C05469=1221.027,359.357,-74.554,-175.932,7.542,148.254
C05470=1221.032,359.109,-74.522,-175.934,7.539,148.254
C05471=1221.036,358.861,-74.489,-175.935,7.537,148.253
C05472=1221.040,358.613,-74.455,-175.937,7.533,148.253
C05473=1221.044,358.365,-74.424,-175.939,7.530,148.253
C05474=1221.048,358.118,-74.390,-175.940,7.528,148.253
C05475=1221.053,357.870,-74.358,-175.941,7.525,148.252
C05476=1221.056,357.622,-74.326,-175.944,7.522,148.252
C05477=1221.061,357.374,-74.293,-175.945,7.519,148.252
C05478=1221.065,357.126,-74.260,-175.947,7.517,148.252
C05479=1221.069,356.878,-74.228,-175.949,7.513,148.251
C05480=1221.073,356.631,-74.195,-175.950,7.510,148.251
C05481=1221.077,356.382,-74.163,-175.952,7.508,148.251
C05482=1221.082,356.135,-74.130,-175.954,7.505,148.251
C05483=1221.086,355.887,-74.098,-175.955,7.502,148.250
C05484=1221.090,355.639,-74.065,-175.957,7.499,148.250
C05485=1221.094,355.391,-74.033,-175.959,7.497,148.250
C05486=1221.098,355.144,-74.000,-175.961,7.493,148.249
C05487=1221.102,354.895,-73.968,-175.962,7.490,148.249
C05488=1221.106,354.648,-73.936,-175.964,7.488,148.249
C05489=1221.110,354.400,-73.903,-175.965,7.485,148.249
C05490=1221.115,354.152,-73.871,-175.967,7.482,148.248
C05491=1221.118,353.905,-73.838,-175.969,7.480,148.248
C05492=1221.123,353.656,-73.806,-175.971,7.477,148.248
C05493=1221.128,353.409,-73.773,-175.972,7.473,148.248
C05494=1221.131,353.161,-73.741,-175.974,7.471,148.247
C05495=1221.136,352.913,-73.708,-175.976,7.468,148.247
C05496=1221.139,352.665,-73.677,-175.978,7.465,148.247
C05497=1221.144,352.417,-73.643,-175.979,7.462,148.247
C05498=1221.148,352.170,-73.612,-175.981,7.460,148.247
C05499=1221.152,351.921,-73.580,-175.983,7.457,148.246
C05500=1221.156,351.674,-73.546,-175.985,7.454,148.246
C05501=1221.160,351.426,-73.515,-175.987,7.452,148.246
C05502=1221.165,351.178,-73.482,-175.988,7.448,148.246
C05503=1221.169,350.930,-73.451,-175.990,7.445,148.245
C05504=1221.173,350.682,-73.417,-175.992,7.443,148.245
C05505=1221.177,350.434,-73.386,-175.994,7.439,148.245
C05506=1221.182,350.186,-73.354,-175.995,7.437,148.245
C05507=1221.185,349.938,-73.322,-175.997,7.434,148.245
C05508=1221.190,349.691,-73.289,-175.999,7.431,148.244
C05509=1221.193,349.443,-73.257,-176.001,7.429,148.244
C05510=1221.198,349.195,-73.225,-176.002,7.426,148.244
C05511=1221.202,348.947,-73.193,-176.005,7.423,148.244
C05512=1221.206,348.699,-73.160,-176.006,7.420,148.244
C05513=1221.210,348.451,-73.128,-176.008,7.418,148.244
C05514=1221.215,348.204,-73.096,-176.010,7.414,148.243
C05515=1221.219,347.955,-73.064,-176.012,7.412,148.243
C05516=1221.223,347.707,-73.031,-176.013,7.409,148.243
C05517=1221.227,347.460,-73.000,-176.016,7.406,148.243
C05518=1221.232,347.211,-72.967,-176.017,7.403,148.243
C05519=1221.236,346.963,-72.936,-176.019,7.401,148.242
C05520=1221.240,346.716,-72.904,-176.021,7.397,148.242
C05521=1221.244,346.468,-72.872,-176.023,7.395,148.242
C05522=1221.248,346.220,-72.840,-176.024,7.392,148.242
C05523=1221.253,345.972,-72.808,-176.027,7.389,148.242
C05524=1221.257,345.724,-72.776,-176.029,7.387,148.242
C05525=1221.260,345.476,-72.744,-176.031,7.383,148.241
C05526=1221.265,345.229,-72.711,-176.032,7.381,148.241
C05527=1221.269,344.981,-72.679,-176.034,7.378,148.241
C05528=1221.274,344.732,-72.648,-176.036,7.375,148.241
C05529=1221.278,344.485,-72.616,-176.038,7.372,148.241
C05530=1221.282,344.237,-72.584,-176.040,7.370,148.240
C05531=1221.286,343.988,-72.552,-176.042,7.367,148.240
C05532=1221.290,343.741,-72.520,-176.043,7.364,148.240
C05533=1221.294,343.493,-72.489,-176.045,7.362,148.240
C05534=1221.299,343.244,-72.456,-176.048,7.358,148.240
C05535=1221.303,342.997,-72.425,-176.049,7.356,148.240
C05536=1221.307,342.749,-72.393,-176.051,7.353,148.239
C05537=1221.312,342.501,-72.361,-176.053,7.350,148.239
C05538=1221.315,342.253,-72.329,-176.055,7.348,148.239
C05539=1221.319,342.005,-72.297,-176.057,7.345,148.239
C05540=1221.324,341.758,-72.265,-176.059,7.342,148.239
C05541=1221.329,341.480,-72.230,-176.061,7.339,148.239
C05542=1221.333,341.202,-72.195,-176.063,7.335,148.238
C05543=1221.338,340.924,-72.158,-176.066,7.333,148.238
C05544=1221.343,340.646,-72.123,-176.068,7.330,148.238
C05545=1221.346,340.398,-72.092,-176.070,7.326,148.238
C05546=1221.351,340.151,-72.060,-176.072,7.324,148.238
C05547=1221.355,339.902,-72.028,-176.074,7.322,148.238
C05548=1221.360,339.654,-71.997,-176.076,7.318,148.238
C05549=1221.363,339.406,-71.965,-176.077,7.316,148.237
C05550=1221.367,339.158,-71.933,-176.079,7.313,148.237
C05551=1221.371,338.911,-71.902,-176.082,7.310,148.237
C05552=1221.376,338.662,-71.870,-176.083,7.308,148.237
C05553=1221.381,338.415,-71.839,-176.086,7.304,148.237
C05554=1221.384,338.167,-71.807,-176.088,7.302,148.237
C05555=1221.389,337.919,-71.776,-176.089,7.299,148.237
C05556=1221.393,337.671,-71.744,-176.091,7.296,148.236
C05557=1221.398,337.423,-71.712,-176.093,7.294,148.236
C05558=1221.402,337.174,-71.681,-176.096,7.291,148.236
C05559=1221.406,336.927,-71.649,-176.097,7.288,148.236
C05560=1221.410,336.679,-71.618,-176.099,7.286,148.236
C05561=1221.414,336.431,-71.587,-176.102,7.282,148.236
C05562=1221.418,336.183,-71.555,-176.103,7.280,148.236
C05563=1221.422,335.935,-71.523,-176.106,7.277,148.236
C05564=1221.426,335.687,-71.492,-176.108,7.274,148.236
C05565=1221.431,335.439,-71.460,-176.109,7.272,148.235
C05566=1221.435,335.191,-71.429,-176.112,7.269,148.235
C05567=1221.439,334.943,-71.397,-176.114,7.266,148.235
C05568=1221.444,334.695,-71.367,-176.116,7.263,148.235
C05569=1221.447,334.447,-71.335,-176.118,7.261,148.235
C05570=1221.452,334.199,-71.304,-176.119,7.258,148.235
C05571=1221.456,333.951,-71.272,-176.122,7.255,148.235
C05572=1221.460,333.703,-71.241,-176.124,7.253,148.235
C05573=1221.465,333.455,-71.210,-176.126,7.249,148.234
C05574=1221.469,333.207,-71.179,-176.128,7.247,148.234
C05575=1221.473,332.959,-71.147,-176.130,7.244,148.234
C05576=1221.477,332.711,-71.116,-176.132,7.241,148.234
C05577=1221.481,332.463,-71.085,-176.134,7.239,148.234
C05578=1221.485,332.215,-71.053,-176.137,7.236,148.234
C05579=1221.490,331.967,-71.022,-176.138,7.233,148.234
C05580=1221.494,331.719,-70.991,-176.140,7.231,148.234
C05581=1221.498,331.471,-70.960,-176.143,7.228,148.234
C05582=1221.503,331.223,-70.929,-176.145,7.225,148.234
C05583=1221.507,330.975,-70.898,-176.147,7.222,148.234
C05584=1221.511,330.727,-70.866,-176.149,7.220,148.234
C05585=1221.515,330.479,-70.835,-176.151,7.217,148.233
C05586=1221.519,330.231,-70.804,-176.153,7.214,148.233
C05587=1221.523,329.983,-70.772,-176.155,7.212,148.233
C05588=1221.528,329.735,-70.742,-176.158,7.209,148.233
C05589=1221.532,329.487,-70.711,-176.159,7.206,148.233
C05590=1221.536,329.239,-70.679,-176.161,7.204,148.233
C05591=1221.541,328.991,-70.648,-176.163,7.201,148.233
C05592=1221.545,328.742,-70.617,-176.166,7.198,148.233
C05593=1221.549,328.494,-70.587,-176.168,7.195,148.233
C05594=1221.553,328.247,-70.555,-176.170,7.193,148.233
C05595=1221.557,327.998,-70.524,-176.172,7.190,148.232
C05596=1221.562,327.750,-70.493,-176.174,7.187,148.233
C05597=1221.566,327.503,-70.463,-176.176,7.185,148.232
C05598=1221.570,327.255,-70.431,-176.178,7.182,148.232
C05599=1221.574,327.007,-70.400,-176.181,7.179,148.232
C05600=1221.579,326.759,-70.369,-176.183,7.176,148.232
C05601=1221.582,326.510,-70.339,-176.185,7.174,148.232
C05602=1221.587,326.262,-70.308,-176.187,7.171,148.232
C05603=1221.592,326.014,-70.277,-176.189,7.168,148.232
C05604=1221.595,325.766,-70.245,-176.191,7.166,148.232
C05605=1221.600,325.518,-70.215,-176.193,7.163,148.232
C05606=1221.603,325.270,-70.184,-176.196,7.161,148.232
C05607=1221.608,325.022,-70.153,-176.197,7.158,148.232
C05608=1221.612,324.774,-70.123,-176.200,7.155,148.232
C05609=1221.617,324.526,-70.092,-176.202,7.153,148.232
C05610=1221.621,324.277,-70.061,-176.204,7.149,148.232
C05611=1221.625,324.030,-70.031,-176.206,7.147,148.232
C05612=1221.630,323.782,-70.000,-176.208,7.145,148.232
C05613=1221.634,323.533,-69.969,-176.211,7.142,148.231
C05614=1221.638,323.285,-69.938,-176.213,7.139,148.231
C05615=1221.642,323.038,-69.908,-176.215,7.136,148.231
C05616=1221.646,322.789,-69.877,-176.217,7.134,148.231
C05617=1221.651,322.541,-69.846,-176.220,7.131,148.231
C05618=1221.655,322.293,-69.816,-176.222,7.129,148.231
C05619=1221.659,322.045,-69.785,-176.223,7.126,148.231
C05620=1221.663,321.797,-69.754,-176.226,7.123,148.231
C05621=1221.668,321.549,-69.723,-176.228,7.121,148.231
C05622=1221.672,321.301,-69.693,-176.231,7.118,148.231
C05623=1221.676,321.053,-69.662,-176.232,7.115,148.231
C05624=1221.680,320.804,-69.631,-176.235,7.113,148.231
C05625=1221.684,320.557,-69.601,-176.237,7.110,148.231
C05626=1221.689,320.309,-69.570,-176.239,7.107,148.231
C05627=1221.693,320.061,-69.539,-176.241,7.104,148.231
C05628=1221.697,319.813,-69.509,-176.244,7.102,148.231
C05629=1221.702,319.564,-69.479,-176.246,7.100,148.231
C05630=1221.705,319.316,-69.448,-176.248,7.097,148.231
C05631=1221.710,319.068,-69.418,-176.250,7.094,148.231
C05632=1221.714,318.820,-69.387,-176.253,7.091,148.231
C05633=1221.718,318.572,-69.356,-176.255,7.089,148.231
C05634=1221.723,318.323,-69.326,-176.257,7.087,148.231
C05635=1221.727,318.076,-69.296,-176.259,7.083,148.231
C05636=1221.731,317.828,-69.265,-176.261,7.081,148.231
C05637=1221.735,317.579,-69.234,-176.264,7.078,148.231
C05638=1221.739,317.332,-69.204,-176.266,7.076,148.231
C05639=1221.744,317.083,-69.174,-176.268,7.073,148.231
C05640=1221.748,316.835,-69.144,-176.270,7.070,148.231
C05641=1221.753,316.587,-69.113,-176.272,7.068,148.231
C05642=1221.756,316.338,-69.083,-176.275,7.065,148.231
C05643=1221.761,316.090,-69.053,-176.277,7.063,148.231
C05644=1221.765,315.843,-69.022,-176.280,7.060,148.231
C05645=1221.770,315.566,-68.989,-176.281,7.057,148.231
C05646=1221.775,315.291,-68.955,-176.284,7.054,148.231
C05647=1221.780,315.015,-68.922,-176.287,7.051,148.231
C05648=1221.784,314.739,-68.888,-176.289,7.048,148.231
C05649=1221.788,314.492,-68.858,-176.291,7.046,148.231
C05650=1221.793,314.243,-68.827,-176.294,7.044,148.231
C05651=1221.796,313.995,-68.797,-176.296,7.041,148.231
C05652=1221.801,313.746,-68.767,-176.298,7.038,148.231
C05653=1221.805,313.499,-68.737,-176.301,7.035,148.231
C05654=1221.810,313.250,-68.707,-176.303,7.033,148.231
C05655=1221.814,313.002,-68.677,-176.305,7.031,148.231
C05656=1221.819,312.754,-68.646,-176.307,7.028,148.231
C05657=1221.823,312.506,-68.616,-176.310,7.025,148.231
C05658=1221.827,312.259,-68.586,-176.312,7.022,148.231
C05659=1221.832,312.010,-68.556,-176.314,7.020,148.231
C05660=1221.835,311.762,-68.526,-176.316,7.018,148.231
C05661=1221.840,311.513,-68.495,-176.319,7.015,148.231
C05662=1221.844,311.265,-68.466,-176.321,7.013,148.231
C05663=1221.848,311.017,-68.436,-176.324,7.010,148.231
C05664=1221.853,310.769,-68.406,-176.326,7.007,148.231
C05665=1221.857,310.521,-68.376,-176.328,7.005,148.231
C05666=1221.861,310.272,-68.346,-176.330,7.002,148.231
C05667=1221.865,310.025,-68.315,-176.332,7.000,148.231
C05668=1221.870,309.776,-68.286,-176.335,6.997,148.231
C05669=1221.874,309.528,-68.256,-176.337,6.994,148.231
C05670=1221.878,309.280,-68.226,-176.339,6.992,148.231
C05671=1221.883,309.032,-68.196,-176.342,6.989,148.231
C05672=1221.887,308.784,-68.166,-176.344,6.987,148.231
C05673=1221.891,308.536,-68.136,-176.346,6.985,148.231
C05674=1221.896,308.287,-68.107,-176.349,6.982,148.231
C05675=1221.900,308.039,-68.077,-176.351,6.979,148.231
C05676=1221.904,307.791,-68.046,-176.354,6.976,148.231
C05677=1221.908,307.543,-68.017,-176.356,6.974,148.231
C05678=1221.913,307.295,-67.988,-176.358,6.972,148.231
C05679=1221.917,307.047,-67.957,-176.360,6.969,148.231
C05680=1221.921,306.798,-67.927,-176.363,6.967,148.231
C05681=1221.926,306.550,-67.898,-176.365,6.964,148.231
C05682=1221.930,306.302,-67.868,-176.367,6.961,148.231
C05683=1221.934,306.054,-67.838,-176.369,6.959,148.231
C05684=1221.939,305.806,-67.808,-176.372,6.956,148.231
C05685=1221.943,305.557,-67.779,-176.374,6.954,148.231
C05686=1221.947,305.309,-67.749,-176.376,6.952,148.231
C05687=1221.951,305.061,-67.720,-176.379,6.949,148.231
C05688=1221.956,304.813,-67.689,-176.381,6.946,148.231
C05689=1221.960,304.565,-67.660,-176.384,6.943,148.231
C05690=1221.964,304.316,-67.630,-176.386,6.941,148.232
C05691=1221.968,304.068,-67.601,-176.388,6.939,148.232
C05692=1221.972,303.820,-67.571,-176.391,6.936,148.232
C05693=1221.977,303.571,-67.541,-176.393,6.934,148.232
C05694=1221.982,303.323,-67.512,-176.395,6.932,148.232
C05695=1221.986,303.075,-67.482,-176.398,6.929,148.232
C05696=1221.990,302.826,-67.453,-176.400,6.927,148.232
C05697=1221.995,302.579,-67.424,-176.403,6.923,148.232
C05698=1221.999,302.331,-67.394,-176.405,6.921,148.232
C05699=1222.003,302.083,-67.364,-176.407,6.919,148.232
C05700=1222.007,301.835,-67.335,-176.410,6.916,148.232
C05701=1222.012,301.586,-67.305,-176.412,6.914,148.232
C05702=1222.016,301.338,-67.275,-176.414,6.912,148.232
C05703=1222.020,301.090,-67.246,-176.417,6.909,148.232
C05704=1222.024,300.841,-67.216,-176.419,6.906,148.232
C05705=1222.029,300.593,-67.187,-176.421,6.904,148.233
C05706=1222.033,300.344,-67.158,-176.424,6.901,148.233
C05707=1222.038,300.097,-67.129,-176.426,6.899,148.233
C05708=1222.042,299.848,-67.100,-176.428,6.897,148.233
C05709=1222.046,299.600,-67.070,-176.431,6.894,148.233
C05710=1222.050,299.352,-67.041,-176.433,6.892,148.233
C05711=1222.055,299.104,-67.011,-176.436,6.889,148.233
C05712=1222.059,298.855,-66.982,-176.438,6.886,148.233
C05713=1222.063,298.607,-66.952,-176.440,6.885,148.233
C05714=1222.068,298.359,-66.923,-176.443,6.881,148.233
C05715=1222.072,298.111,-66.894,-176.445,6.879,148.233
C05716=1222.076,297.862,-66.865,-176.447,6.877,148.233
C05717=1222.081,297.614,-66.836,-176.450,6.874,148.233
C05718=1222.085,297.366,-66.806,-176.452,6.872,148.233
C05719=1222.089,297.117,-66.777,-176.454,6.870,148.233
C05720=1222.094,296.870,-66.748,-176.457,6.867,148.234
C05721=1222.098,296.621,-66.719,-176.459,6.865,148.234
C05722=1222.102,296.373,-66.689,-176.462,6.862,148.234
C05723=1222.107,296.124,-66.660,-176.464,6.859,148.234
C05724=1222.111,295.876,-66.630,-176.466,6.857,148.234
C05725=1222.115,295.628,-66.603,-176.469,6.855,148.234
C05726=1222.119,295.380,-66.573,-176.472,6.852,148.234
C05727=1222.124,295.132,-66.544,-176.474,6.850,148.234
C05728=1222.128,294.884,-66.514,-176.476,6.848,148.234
C05729=1222.132,294.635,-66.486,-176.478,6.845,148.234
C05730=1222.137,294.387,-66.456,-176.481,6.843,148.235
C05731=1222.141,294.139,-66.427,-176.483,6.841,148.235
C05732=1222.146,293.890,-66.398,-176.486,6.838,148.235
C05733=1222.149,293.642,-66.369,-176.488,6.835,148.235
C05734=1222.154,293.394,-66.340,-176.490,6.833,148.235
C05735=1222.158,293.146,-66.312,-176.493,6.830,148.235
C05736=1222.163,292.897,-66.282,-176.495,6.828,148.235
C05737=1222.167,292.648,-66.253,-176.497,6.826,148.235
C05738=1222.172,292.401,-66.224,-176.500,6.823,148.235
C05739=1222.175,292.153,-66.195,-176.503,6.821,148.235
C05740=1222.180,291.904,-66.167,-176.505,6.819,148.235
C05741=1222.184,291.656,-66.137,-176.507,6.816,148.235
C05742=1222.189,291.408,-66.109,-176.510,6.814,148.236
C05743=1222.193,291.159,-66.079,-176.512,6.812,148.236
C05744=1222.197,290.911,-66.051,-176.515,6.809,148.236
C05745=1222.202,290.663,-66.022,-176.517,6.806,148.236
C05746=1222.206,290.414,-65.993,-176.519,6.804,148.236
C05747=1222.210,290.166,-65.964,-176.522,6.802,148.236
C05748=1222.215,289.918,-65.936,-176.524,6.799,148.236
C05749=1222.220,289.644,-65.905,-176.527,6.796,148.236
C05750=1222.224,289.370,-65.872,-176.530,6.794,148.237
C05751=1222.229,289.096,-65.841,-176.532,6.791,148.237
C05752=1222.234,288.821,-65.809,-176.535,6.789,148.237
C05753=1222.238,288.573,-65.780,-176.538,6.786,148.237
C05754=1222.243,288.325,-65.751,-176.540,6.784,148.237
C05755=1222.247,288.076,-65.723,-176.542,6.782,148.237
C05756=1222.251,287.828,-65.694,-176.545,6.779,148.237
C05757=1222.256,287.580,-65.665,-176.547,6.777,148.237
C05758=1222.260,287.331,-65.637,-176.549,6.775,148.237
C05759=1222.264,287.083,-65.608,-176.552,6.772,148.238
C05760=1222.269,286.835,-65.579,-176.554,6.770,148.238
C05761=1222.273,286.586,-65.551,-176.557,6.768,148.238
C05762=1222.277,286.339,-65.522,-176.559,6.766,148.238
C05763=1222.282,286.090,-65.493,-176.562,6.763,148.238
C05764=1222.286,285.841,-65.465,-176.564,6.761,148.238
C05765=1222.291,285.594,-65.436,-176.567,6.759,148.238
C05766=1222.294,285.345,-65.408,-176.569,6.756,148.238
C05767=1222.299,285.096,-65.379,-176.571,6.753,148.238
C05768=1222.304,284.848,-65.351,-176.574,6.751,148.239
C05769=1222.308,284.599,-65.323,-176.576,6.749,148.239
C05770=1222.312,284.352,-65.294,-176.579,6.746,148.239
C05771=1222.316,284.103,-65.265,-176.581,6.744,148.239
C05772=1222.321,283.855,-65.237,-176.583,6.742,148.239
C05773=1222.325,283.606,-65.209,-176.586,6.739,148.239
C05774=1222.329,283.358,-65.180,-176.589,6.737,148.240
C05775=1222.334,283.110,-65.151,-176.591,6.735,148.240
C05776=1222.338,282.861,-65.123,-176.593,6.733,148.240
C05777=1222.343,282.613,-65.095,-176.596,6.730,148.240
C05778=1222.347,282.365,-65.066,-176.598,6.728,148.240
C05779=1222.352,282.116,-65.038,-176.601,6.726,148.240
C05780=1222.356,281.868,-65.010,-176.603,6.724,148.240
C05781=1222.361,281.620,-64.981,-176.606,6.721,148.240
C05782=1222.364,281.371,-64.953,-176.608,6.719,148.241
C05783=1222.370,281.123,-64.925,-176.610,6.717,148.241
C05784=1222.373,280.874,-64.897,-176.613,6.714,148.241
C05785=1222.377,280.626,-64.869,-176.616,6.712,148.241
C05786=1222.382,280.378,-64.840,-176.618,6.709,148.241
C05787=1222.386,280.129,-64.812,-176.620,6.708,148.241
C05788=1222.391,279.881,-64.784,-176.623,6.705,148.241
C05789=1222.395,279.632,-64.756,-176.626,6.703,148.242
C05790=1222.400,279.384,-64.727,-176.628,6.700,148.242
C05791=1222.404,279.135,-64.699,-176.630,6.698,148.242
C05792=1222.408,278.888,-64.671,-176.633,6.695,148.242
C05793=1222.412,278.639,-64.643,-176.635,6.693,148.242
C05794=1222.417,278.391,-64.615,-176.638,6.691,148.242
C05795=1222.421,278.142,-64.586,-176.640,6.689,148.243
C05796=1222.426,277.894,-64.558,-176.643,6.686,148.243
C05797=1222.430,277.646,-64.531,-176.645,6.684,148.243
C05798=1222.434,277.397,-64.502,-176.647,6.682,148.243
C05799=1222.439,277.149,-64.474,-176.650,6.680,148.243
C05800=1222.443,276.901,-64.446,-176.652,6.677,148.243
C05801=1222.448,276.652,-64.418,-176.655,6.675,148.244
C05802=1222.452,276.403,-64.390,-176.657,6.673,148.244
C05803=1222.456,276.156,-64.362,-176.660,6.671,148.244
C05804=1222.461,275.907,-64.334,-176.662,6.669,148.244
C05805=1222.465,275.659,-64.306,-176.665,6.666,148.244
C05806=1222.469,275.411,-64.278,-176.667,6.664,148.244
C05807=1222.474,275.161,-64.250,-176.670,6.662,148.245
C05808=1222.478,274.914,-64.222,-176.672,6.660,148.245
C05809=1222.482,274.665,-64.194,-176.675,6.657,148.245
C05810=1222.486,274.417,-64.166,-176.677,6.655,148.245
C05811=1222.491,274.168,-64.138,-176.679,6.653,148.245
C05812=1222.496,273.920,-64.111,-176.682,6.651,148.245
C05813=1222.500,273.672,-64.083,-176.685,6.648,148.245
C05814=1222.504,273.423,-64.055,-176.687,6.646,148.246
C05815=1222.509,273.175,-64.027,-176.689,6.644,148.246
C05816=1222.513,272.927,-63.999,-176.692,6.642,148.246
C05817=1222.517,272.678,-63.971,-176.694,6.640,148.246
C05818=1222.522,272.430,-63.944,-176.697,6.637,148.246
C05819=1222.526,272.181,-63.916,-176.699,6.635,148.246
C05820=1222.531,271.933,-63.887,-176.702,6.633,148.247
C05821=1222.535,271.684,-63.860,-176.704,6.631,148.247
C05822=1222.539,271.436,-63.832,-176.707,6.629,148.247
C05823=1222.544,271.187,-63.805,-176.709,6.626,148.247
C05824=1222.548,270.939,-63.777,-176.712,6.624,148.247
C05825=1222.553,270.690,-63.749,-176.714,6.622,148.247
C05826=1222.557,270.442,-63.722,-176.717,6.620,148.248
C05827=1222.562,270.194,-63.694,-176.719,6.618,148.248
C05828=1222.566,269.945,-63.666,-176.722,6.615,148.248
C05829=1222.570,269.697,-63.639,-176.724,6.613,148.248
C05830=1222.575,269.449,-63.612,-176.727,6.611,148.248
C05831=1222.578,269.200,-63.583,-176.729,6.609,148.249
C05832=1222.583,268.951,-63.556,-176.731,6.607,148.249
C05833=1222.588,268.703,-63.528,-176.735,6.604,148.249
C05834=1222.592,268.454,-63.501,-176.737,6.602,148.249
C05835=1222.597,268.206,-63.473,-176.739,6.600,148.249
C05836=1222.601,267.958,-63.446,-176.741,6.598,148.250
C05837=1222.606,267.710,-63.418,-176.744,6.596,148.250
C05838=1222.610,267.461,-63.391,-176.747,6.593,148.250
C05839=1222.614,267.212,-63.363,-176.749,6.591,148.250
C05840=1222.619,266.964,-63.336,-176.751,6.589,148.250
C05841=1222.623,266.716,-63.309,-176.754,6.587,148.251
C05842=1222.627,266.467,-63.280,-176.756,6.585,148.251
C05843=1222.632,266.219,-63.253,-176.759,6.583,148.251
C05844=1222.636,265.970,-63.226,-176.762,6.580,148.251
C05845=1222.641,265.722,-63.199,-176.764,6.578,148.251
C05846=1222.645,265.473,-63.171,-176.767,6.576,148.252
C05847=1222.649,265.225,-63.144,-176.769,6.574,148.252
C05848=1222.654,264.977,-63.116,-176.771,6.572,148.252
C05849=1222.658,264.728,-63.089,-176.773,6.570,148.252
C05850=1222.663,264.479,-63.062,-176.777,6.567,148.252
C05851=1222.667,264.231,-63.034,-176.779,6.565,148.253
C05852=1222.672,263.983,-63.007,-176.781,6.563,148.253
C05853=1222.677,263.710,-62.977,-176.784,6.561,148.253
C05854=1222.682,263.437,-62.948,-176.787,6.558,148.253
C05855=1222.686,263.165,-62.918,-176.789,6.556,148.253
C05856=1222.691,262.891,-62.887,-176.792,6.553,148.254
C05857=1222.695,262.643,-62.860,-176.795,6.551,148.254
C05858=1222.700,262.395,-62.832,-176.797,6.549,148.254
C05859=1222.704,262.147,-62.805,-176.800,6.547,148.254
C05860=1222.709,261.898,-62.778,-176.802,6.545,148.255
C05861=1222.712,261.649,-62.751,-176.804,6.543,148.255
C05862=1222.717,261.401,-62.724,-176.808,6.540,148.255
C05863=1222.722,261.152,-62.697,-176.810,6.538,148.255
C05864=1222.726,260.904,-62.670,-176.812,6.536,148.255
C05865=1222.731,260.656,-62.643,-176.815,6.534,148.256
C05866=1222.735,260.407,-62.615,-176.817,6.532,148.256
C05867=1222.740,260.159,-62.588,-176.820,6.530,148.256
C05868=1222.743,259.910,-62.562,-176.822,6.528,148.256
C05869=1222.748,259.662,-62.535,-176.825,6.526,148.256
C05870=1222.753,259.413,-62.507,-176.828,6.524,148.257
C05871=1222.757,259.165,-62.480,-176.830,6.521,148.257
C05872=1222.762,258.916,-62.453,-176.832,6.520,148.257
C05873=1222.766,258.668,-62.427,-176.835,6.518,148.257
C05874=1222.771,258.419,-62.400,-176.837,6.515,148.257
C05875=1222.775,258.171,-62.373,-176.840,6.514,148.258
C05876=1222.779,257.922,-62.345,-176.842,6.512,148.258
C05877=1222.784,257.673,-62.318,-176.845,6.509,148.258
C05878=1222.788,257.425,-62.292,-176.848,6.507,148.258
C05879=1222.793,257.176,-62.265,-176.850,6.505,148.258
C05880=1222.797,256.928,-62.238,-176.852,6.503,148.259
C05881=1222.802,256.679,-62.211,-176.855,6.501,148.259
C05882=1222.806,256.431,-62.184,-176.857,6.499,148.259
C05883=1222.810,256.183,-62.157,-176.860,6.497,148.259
C05884=1222.815,255.934,-62.130,-176.862,6.495,148.260
C05885=1222.820,255.686,-62.103,-176.865,6.492,148.260
C05886=1222.824,255.438,-62.076,-176.868,6.490,148.260
C05887=1222.829,255.189,-62.050,-176.870,6.488,148.260
C05888=1222.833,254.939,-62.023,-176.872,6.486,148.260
C05889=1222.837,254.691,-61.996,-176.875,6.484,148.261
C05890=1222.841,254.443,-61.969,-176.878,6.482,148.261
C05891=1222.846,254.194,-61.942,-176.880,6.480,148.261
C05892=1222.850,253.946,-61.916,-176.882,6.478,148.261
C05893=1222.855,253.697,-61.889,-176.885,6.476,148.262
C05894=1222.859,253.448,-61.862,-176.887,6.474,148.262
C05895=1222.863,253.200,-61.836,-176.890,6.472,148.262
C05896=1222.868,252.952,-61.809,-176.893,6.469,148.262
C05897=1222.872,252.703,-61.783,-176.895,6.467,148.262
C05898=1222.877,252.454,-61.756,-176.898,6.465,148.263
C05899=1222.882,252.206,-61.729,-176.900,6.463,148.263
C05900=1222.885,251.958,-61.702,-176.903,6.462,148.263
C05901=1222.890,251.709,-61.676,-176.905,6.459,148.263
C05902=1222.894,251.460,-61.650,-176.908,6.457,148.264
C05903=1222.899,251.212,-61.622,-176.910,6.456,148.264
C05904=1222.904,250.963,-61.596,-176.912,6.453,148.264
C05905=1222.908,250.715,-61.570,-176.915,6.452,148.264
C05906=1222.913,250.466,-61.543,-176.917,6.450,148.265
C05907=1222.917,250.217,-61.517,-176.920,6.447,148.265
C05908=1222.921,249.969,-61.490,-176.923,6.445,148.265
C05909=1222.925,249.721,-61.463,-176.925,6.443,148.265
C05910=1222.930,249.471,-61.437,-176.928,6.441,148.266
C05911=1222.935,249.224,-61.411,-176.930,6.439,148.266
C05912=1222.939,248.976,-61.384,-176.933,6.437,148.266
C05913=1222.944,248.727,-61.358,-176.935,6.435,148.266
C05914=1222.948,248.478,-61.331,-176.938,6.433,148.267
C05915=1222.953,248.229,-61.305,-176.940,6.431,148.267
C05916=1222.957,247.981,-61.278,-176.943,6.429,148.267
C05917=1222.961,247.732,-61.252,-176.945,6.427,148.267
C05918=1222.966,247.484,-61.225,-176.947,6.425,148.268
C05919=1222.970,247.235,-61.200,-176.950,6.423,148.268
C05920=1222.975,246.986,-61.173,-176.953,6.421,148.268
C05921=1222.979,246.738,-61.147,-176.955,6.419,148.269
C05922=1222.984,246.489,-61.120,-176.957,6.417,148.269
C05923=1222.988,246.240,-61.094,-176.960,6.415,148.269
C05924=1222.993,245.993,-61.068,-176.963,6.413,148.269
C05925=1222.998,245.744,-61.042,-176.966,6.411,148.269
C05926=1223.002,245.495,-61.015,-176.968,6.409,148.270
C05927=1223.006,245.246,-60.989,-176.971,6.407,148.270
C05928=1223.010,244.998,-60.962,-176.973,6.405,148.270
C05929=1223.015,244.749,-60.937,-176.976,6.403,148.271
C05930=1223.020,244.500,-60.910,-176.978,6.401,148.271
C05931=1223.024,244.252,-60.884,-176.981,6.399,148.271
C05932=1223.028,244.004,-60.858,-176.983,6.397,148.271
C05933=1223.033,243.755,-60.832,-176.986,6.395,148.272
C05934=1223.037,243.507,-60.806,-176.988,6.393,148.272
C05935=1223.042,243.258,-60.779,-176.991,6.391,148.272
C05936=1223.046,243.009,-60.753,-176.993,6.389,148.272
C05937=1223.050,242.761,-60.727,-176.996,6.387,148.273
C05938=1223.055,242.512,-60.702,-176.998,6.385,148.273
C05939=1223.060,242.263,-60.675,-177.001,6.383,148.273
C05940=1223.064,242.015,-60.649,-177.003,6.381,148.273
C05941=1223.068,241.766,-60.623,-177.006,6.380,148.274
C05942=1223.073,241.517,-60.597,-177.008,6.378,148.274
C05943=1223.077,241.268,-60.571,-177.011,6.375,148.274
C05944=1223.082,241.021,-60.545,-177.013,6.374,148.274
C05945=1223.087,240.772,-60.518,-177.016,6.372,148.275
C05946=1223.091,240.523,-60.493,-177.018,6.370,148.275
C05947=1223.095,240.274,-60.467,-177.021,6.368,148.275
C05948=1223.100,240.026,-60.442,-177.023,6.366,148.275
C05949=1223.105,239.778,-60.415,-177.026,6.364,148.276
C05950=1223.109,239.529,-60.389,-177.028,6.362,148.276
C05951=1223.113,239.280,-60.363,-177.031,6.360,148.276
C05952=1223.118,239.031,-60.337,-177.034,6.358,148.277
C05953=1223.122,238.783,-60.312,-177.036,6.356,148.277
C05954=1223.127,238.534,-60.286,-177.038,6.354,148.277
C05955=1223.131,238.286,-60.259,-177.041,6.352,148.277
C05956=1223.135,238.037,-60.233,-177.044,6.351,148.278
C05957=1223.141,237.766,-60.206,-177.047,6.348,148.278
C05958=1223.145,237.494,-60.178,-177.049,6.346,148.278
C05959=1223.150,237.223,-60.149,-177.052,6.344,148.279
C05960=1223.155,236.951,-60.121,-177.055,6.342,148.279
C05961=1223.159,236.703,-60.095,-177.057,6.340,148.279
C05962=1223.165,236.454,-60.069,-177.059,6.338,148.279
C05963=1223.169,236.205,-60.044,-177.062,6.336,148.280
C05964=1223.173,235.957,-60.018,-177.065,6.334,148.280
C05965=1223.178,235.708,-59.993,-177.067,6.333,148.280
C05966=1223.182,235.460,-59.967,-177.070,6.331,148.281
C05967=1223.187,235.211,-59.941,-177.073,6.329,148.281
C05968=1223.191,234.962,-59.915,-177.075,6.327,148.281
C05969=1223.196,234.714,-59.890,-177.077,6.325,148.281
C05970=1223.200,234.465,-59.864,-177.080,6.323,148.282
C05971=1223.205,234.216,-59.838,-177.083,6.321,148.282
C05972=1223.210,233.968,-59.812,-177.085,6.319,148.282
C05973=1223.214,233.719,-59.787,-177.088,6.317,148.283
C05974=1223.218,233.470,-59.761,-177.090,6.315,148.283
C05975=1223.223,233.222,-59.736,-177.093,6.313,148.283
C05976=1223.228,232.973,-59.711,-177.095,6.311,148.283
C05977=1223.232,232.724,-59.685,-177.098,6.309,148.284
C05978=1223.237,232.476,-59.659,-177.100,6.308,148.284
C05979=1223.241,232.227,-59.634,-177.103,6.306,148.284
C05980=1223.245,231.978,-59.608,-177.106,6.304,148.285
C05981=1223.250,231.730,-59.583,-177.108,6.302,148.285
C05982=1223.254,231.481,-59.557,-177.110,6.300,148.285
C05983=1223.259,231.233,-59.532,-177.113,6.298,148.285
C05984=1223.263,230.984,-59.506,-177.116,6.296,148.286
C05985=1223.268,230.735,-59.481,-177.118,6.294,148.286
C05986=1223.272,230.487,-59.455,-177.121,6.292,148.286
C05987=1223.277,230.237,-59.430,-177.124,6.290,148.287
C05988=1223.282,229.989,-59.405,-177.126,6.289,148.287
C05989=1223.286,229.741,-59.379,-177.128,6.286,148.287
C05990=1223.290,229.492,-59.353,-177.131,6.285,148.287
C05991=1223.295,229.243,-59.329,-177.134,6.283,148.288
C05992=1223.299,228.995,-59.303,-177.136,6.281,148.288
C05993=1223.304,228.746,-59.278,-177.139,6.279,148.288
C05994=1223.308,228.497,-59.253,-177.141,6.278,148.289
C05995=1223.312,228.248,-59.227,-177.143,6.276,148.289
C05996=1223.317,228.000,-59.202,-177.146,6.274,148.289
C05997=1223.322,227.751,-59.177,-177.149,6.272,148.290
C05998=1223.327,227.503,-59.151,-177.151,6.270,148.290
C05999=1223.331,227.254,-59.126,-177.154,6.268,148.290
C06000=1223.336,227.005,-59.101,-177.156,6.266,148.290
C06001=1223.340,226.757,-59.076,-177.159,6.265,148.291
C06002=1223.344,226.508,-59.051,-177.161,6.263,148.291
C06003=1223.349,226.259,-59.025,-177.164,6.261,148.291
C06004=1223.353,226.010,-59.000,-177.167,6.259,148.292
C06005=1223.358,225.762,-58.975,-177.169,6.257,148.292
C06006=1223.362,225.513,-58.949,-177.172,6.255,148.292
C06007=1223.367,225.264,-58.925,-177.175,6.253,148.293
C06008=1223.371,225.015,-58.899,-177.177,6.252,148.293
C06009=1223.376,224.767,-58.875,-177.179,6.249,148.293
C06010=1223.380,224.518,-58.849,-177.182,6.247,148.293
C06011=1223.386,224.269,-58.824,-177.185,6.246,148.294
C06012=1223.389,224.021,-58.799,-177.187,6.245,148.294
C06013=1223.394,223.772,-58.775,-177.189,6.243,148.294
C06014=1223.398,223.523,-58.749,-177.192,6.241,148.295
C06015=1223.404,223.274,-58.724,-177.194,6.239,148.295
C06016=1223.407,223.026,-58.699,-177.197,6.237,148.295
C06017=1223.412,222.777,-58.674,-177.200,6.235,148.296
C06018=1223.416,222.528,-58.649,-177.202,6.233,148.296
C06019=1223.422,222.280,-58.624,-177.205,6.232,148.296
C06020=1223.426,222.031,-58.600,-177.208,6.230,148.297
C06021=1223.430,221.783,-58.574,-177.210,6.228,148.297
C06022=1223.435,221.534,-58.549,-177.213,6.226,148.297
C06023=1223.439,221.285,-58.524,-177.216,6.224,148.298
C06024=1223.444,221.037,-58.500,-177.218,6.222,148.298
C06025=1223.448,220.787,-58.475,-177.220,6.221,148.298
C06026=1223.452,220.539,-58.450,-177.222,6.219,148.299
C06027=1223.457,220.290,-58.425,-177.225,6.217,148.299
C06028=1223.462,220.041,-58.400,-177.228,6.215,148.299
C06029=1223.466,219.793,-58.375,-177.230,6.213,148.300
C06030=1223.471,219.544,-58.350,-177.233,6.212,148.300
C06031=1223.476,219.295,-58.326,-177.236,6.210,148.300
C06032=1223.480,219.046,-58.301,-177.238,6.208,148.300
C06033=1223.485,218.798,-58.276,-177.241,6.206,148.301
C06034=1223.489,218.549,-58.251,-177.243,6.204,148.301
C06035=1223.493,218.300,-58.227,-177.246,6.202,148.301
C06036=1223.499,218.052,-58.202,-177.249,6.200,148.302
C06037=1223.502,217.803,-58.177,-177.251,6.199,148.302
C06038=1223.507,217.554,-58.152,-177.253,6.198,148.303
C06039=1223.512,217.306,-58.127,-177.256,6.196,148.303
C06040=1223.516,217.056,-58.103,-177.259,6.194,148.303
C06041=1223.521,216.808,-58.078,-177.261,6.192,148.303
C06042=1223.525,216.559,-58.053,-177.264,6.190,148.304
C06043=1223.530,216.311,-58.029,-177.267,6.188,148.304
C06044=1223.534,216.062,-58.004,-177.269,6.186,148.304
C06045=1223.539,215.813,-57.979,-177.272,6.185,148.305
C06046=1223.543,215.564,-57.955,-177.274,6.183,148.305
C06047=1223.548,215.316,-57.931,-177.276,6.182,148.306
C06048=1223.553,215.066,-57.906,-177.279,6.180,148.306
C06049=1223.557,214.818,-57.882,-177.282,6.178,148.306
C06050=1223.562,214.570,-57.856,-177.284,6.176,148.307
C06051=1223.566,214.320,-57.832,-177.287,6.174,148.307
C06052=1223.571,214.072,-57.807,-177.290,6.172,148.307
C06053=1223.575,213.823,-57.783,-177.292,6.171,148.308
C06054=1223.579,213.574,-57.759,-177.295,6.169,148.308
C06055=1223.584,213.326,-57.734,-177.298,6.167,148.308
C06056=1223.589,213.077,-57.710,-177.300,6.166,148.309
C06057=1223.594,212.828,-57.685,-177.302,6.164,148.309
C06058=1223.598,212.579,-57.661,-177.305,6.162,148.309
C06059=1223.603,212.331,-57.636,-177.308,6.160,148.310
C06060=1223.607,212.082,-57.612,-177.310,6.158,148.310
C06061=1223.612,211.811,-57.586,-177.313,6.157,148.310
C06062=1223.617,211.540,-57.559,-177.315,6.155,148.311
C06063=1223.622,211.270,-57.532,-177.319,6.153,148.311
C06064=1223.627,211.000,-57.506,-177.321,6.151,148.311
C06065=1223.632,210.752,-57.481,-177.324,6.149,148.312
C06066=1223.636,210.503,-57.457,-177.326,6.148,148.312
C06067=1223.641,210.253,-57.433,-177.329,6.146,148.312
C06068=1223.645,210.005,-57.409,-177.332,6.144,148.313
C06069=1223.650,209.756,-57.385,-177.334,6.142,148.313
C06070=1223.654,209.507,-57.360,-177.337,6.140,148.313
C06071=1223.659,209.259,-57.336,-177.340,6.138,148.314
C06072=1223.663,209.010,-57.312,-177.342,6.137,148.314
C06073=1223.668,208.761,-57.287,-177.344,6.136,148.314
C06074=1223.672,208.512,-57.263,-177.347,6.134,148.315
C06075=1223.677,208.263,-57.239,-177.350,6.132,148.315
C06076=1223.682,208.015,-57.215,-177.352,6.130,148.315
C06077=1223.686,207.766,-57.190,-177.355,6.128,148.316
C06078=1223.691,207.518,-57.166,-177.357,6.127,148.316
C06079=1223.696,207.268,-57.142,-177.360,6.125,148.317
C06080=1223.700,207.019,-57.118,-177.362,6.123,148.317
C06081=1223.704,206.771,-57.094,-177.365,6.122,148.317
C06082=1223.709,206.522,-57.070,-177.367,6.120,148.318
C06083=1223.714,206.273,-57.046,-177.370,6.118,148.318
C06084=1223.718,206.024,-57.021,-177.373,6.116,148.318
C06085=1223.722,205.776,-56.997,-177.375,6.115,148.319
C06086=1223.728,205.526,-56.973,-177.378,6.113,148.319
C06087=1223.732,205.278,-56.949,-177.381,6.112,148.319
C06088=1223.737,205.029,-56.925,-177.383,6.110,148.320
C06089=1223.741,204.780,-56.902,-177.386,6.108,148.320
C06090=1223.745,204.531,-56.877,-177.388,6.107,148.321
C06091=1223.750,204.283,-56.853,-177.391,6.105,148.321
C06092=1223.755,204.034,-56.829,-177.393,6.103,148.321
C06093=1223.759,203.785,-56.805,-177.396,6.101,148.322
C06094=1223.764,203.536,-56.782,-177.399,6.099,148.322
C06095=1223.768,203.288,-56.758,-177.401,6.098,148.322
C06096=1223.774,203.039,-56.733,-177.403,6.097,148.323
C06097=1223.778,202.790,-56.710,-177.406,6.095,148.323
C06098=1223.782,202.541,-56.685,-177.409,6.093,148.323
C06099=1223.787,202.292,-56.662,-177.412,6.091,148.324
C06100=1223.791,202.043,-56.638,-177.414,6.090,148.324
C06101=1223.796,201.794,-56.615,-177.416,6.089,148.325
C06102=1223.800,201.546,-56.591,-177.419,6.087,148.325
C06103=1223.806,201.297,-56.567,-177.422,6.085,148.325
C06104=1223.810,201.048,-56.543,-177.424,6.083,148.326
C06105=1223.815,200.799,-56.519,-177.427,6.081,148.326
C06106=1223.819,200.551,-56.495,-177.429,6.080,148.326
C06107=1223.824,200.302,-56.472,-177.432,6.078,148.327
C06108=1223.828,200.053,-56.447,-177.434,6.076,148.327
C06109=1223.832,199.804,-56.424,-177.437,6.075,148.327
C06110=1223.837,199.555,-56.400,-177.440,6.073,148.328
C06111=1223.841,199.306,-56.377,-177.442,6.072,148.328
C06112=1223.846,199.058,-56.352,-177.445,6.070,148.329
C06113=1223.851,198.809,-56.329,-177.447,6.068,148.329
C06114=1223.855,198.560,-56.306,-177.450,6.066,148.329
C06115=1223.860,198.311,-56.282,-177.453,6.065,148.330
C06116=1223.864,198.062,-56.258,-177.455,6.064,148.330
C06117=1223.869,197.813,-56.235,-177.457,6.062,148.330
C06118=1223.873,197.565,-56.211,-177.460,6.060,148.331
C06119=1223.879,197.315,-56.187,-177.463,6.058,148.331
C06120=1223.883,197.067,-56.163,-177.465,6.057,148.332
C06121=1223.888,196.818,-56.139,-177.468,6.056,148.332
C06122=1223.892,196.569,-56.117,-177.471,6.054,148.332
C06123=1223.897,196.320,-56.093,-177.473,6.052,148.333
C06124=1223.901,196.072,-56.069,-177.476,6.050,148.333
C06125=1223.906,195.823,-56.046,-177.478,6.049,148.333
C06126=1223.910,195.574,-56.023,-177.481,6.047,148.334
C06127=1223.915,195.325,-55.998,-177.483,6.045,148.334
C06128=1223.920,195.076,-55.975,-177.486,6.043,148.334
C06129=1223.924,194.827,-55.952,-177.488,6.043,148.335
C06130=1223.929,194.578,-55.928,-177.491,6.041,148.335
C06131=1223.934,194.329,-55.905,-177.494,6.039,148.336
C06132=1223.938,194.081,-55.881,-177.496,6.037,148.336
C06133=1223.943,193.832,-55.858,-177.498,6.036,148.336
C06134=1223.947,193.583,-55.834,-177.501,6.034,148.337
C06135=1223.952,193.334,-55.811,-177.504,6.033,148.337
C06136=1223.957,193.085,-55.788,-177.507,6.031,148.338
C06137=1223.961,192.836,-55.763,-177.509,6.030,148.338
C06138=1223.965,192.588,-55.741,-177.512,6.028,148.338
C06139=1223.970,192.338,-55.717,-177.514,6.026,148.339
C06140=1223.975,192.090,-55.694,-177.517,6.025,148.339
C06141=1223.980,191.841,-55.671,-177.519,6.024,148.339
C06142=1223.985,191.592,-55.648,-177.522,6.022,148.340
C06143=1223.989,191.343,-55.624,-177.524,6.020,148.340
C06144=1223.994,191.094,-55.601,-177.527,6.018,148.341
C06145=1223.998,190.845,-55.578,-177.529,6.017,148.341
C06146=1224.003,190.596,-55.555,-177.532,6.015,148.341
C06147=1224.007,190.347,-55.531,-177.535,6.014,148.342
C06148=1224.012,190.099,-55.507,-177.537,6.012,148.342
C06149=1224.016,189.850,-55.484,-177.539,6.011,148.343
C06150=1224.021,189.602,-55.462,-177.543,6.009,148.343
C06151=1224.026,189.353,-55.438,-177.545,6.007,148.343
C06152=1224.030,189.104,-55.415,-177.547,6.006,148.344
C06153=1224.035,188.855,-55.392,-177.550,6.005,148.344
C06154=1224.040,188.606,-55.368,-177.553,6.003,148.345
C06155=1224.044,188.356,-55.346,-177.555,6.001,148.345
C06156=1224.049,188.107,-55.323,-177.558,6.000,148.345
C06157=1224.053,187.858,-55.299,-177.560,5.998,148.346
C06158=1224.059,187.610,-55.276,-177.563,5.997,148.346
C06159=1224.063,187.361,-55.254,-177.565,5.996,148.347
C06160=1224.067,187.112,-55.230,-177.568,5.994,148.347
C06161=1224.072,186.863,-55.207,-177.571,5.992,148.347
C06162=1224.076,186.614,-55.184,-177.574,5.990,148.348
C06163=1224.081,186.365,-55.161,-177.576,5.989,148.348
C06164=1224.086,186.117,-55.138,-177.578,5.988,148.349
C06165=1224.090,185.847,-55.113,-177.581,5.986,148.349
C06166=1224.095,185.577,-55.088,-177.584,5.984,148.349
C06167=1224.101,185.307,-55.063,-177.587,5.982,148.350
C06168=1224.105,185.038,-55.039,-177.589,5.980,148.350
C06169=1224.111,184.790,-55.016,-177.592,5.980,148.351
C06170=1224.115,184.541,-54.992,-177.595,5.978,148.351
C06171=1224.120,184.291,-54.970,-177.597,5.976,148.352
C06172=1224.124,184.042,-54.947,-177.599,5.975,148.352
C06173=1224.129,183.793,-54.923,-177.602,5.973,148.352
C06174=1224.134,183.545,-54.901,-177.605,5.972,148.353
C06175=1224.138,183.296,-54.878,-177.608,5.970,148.353
C06176=1224.142,183.047,-54.856,-177.610,5.969,148.354
C06177=1224.147,182.798,-54.832,-177.613,5.967,148.354
C06178=1224.152,182.549,-54.809,-177.615,5.965,148.354
C06179=1224.156,182.301,-54.786,-177.617,5.964,148.355
C06180=1224.161,182.051,-54.764,-177.620,5.963,148.355
C06181=1224.165,181.802,-54.741,-177.623,5.961,148.356
C06182=1224.170,181.553,-54.718,-177.625,5.960,148.356
C06183=1224.176,181.304,-54.695,-177.628,5.958,148.356
C06184=1224.180,181.056,-54.673,-177.631,5.957,148.357
C06185=1224.184,180.807,-54.649,-177.633,5.956,148.357
C06186=1224.189,180.557,-54.627,-177.636,5.954,148.358
C06187=1224.194,180.309,-54.604,-177.638,5.952,148.358
C06188=1224.198,180.060,-54.582,-177.640,5.951,148.358
C06189=1224.203,179.810,-54.559,-177.644,5.949,148.359
C06190=1224.207,179.562,-54.536,-177.646,5.948,148.359
C06191=1224.212,179.313,-54.514,-177.648,5.947,148.360
C06192=1224.216,179.064,-54.491,-177.651,5.945,148.360
C06193=1224.221,178.814,-54.468,-177.654,5.943,148.360
C06194=1224.226,178.566,-54.446,-177.656,5.942,148.361
C06195=1224.231,178.317,-54.423,-177.659,5.940,148.361
C06196=1224.235,178.068,-54.401,-177.662,5.939,148.362
C06197=1224.240,177.820,-54.378,-177.664,5.938,148.362
C06198=1224.245,177.570,-54.356,-177.667,5.936,148.363
C06199=1224.249,177.321,-54.332,-177.669,5.934,148.363
C06200=1224.254,177.073,-54.311,-177.672,5.933,148.363
C06201=1224.258,176.824,-54.288,-177.674,5.931,148.364
C06202=1224.263,176.574,-54.265,-177.677,5.931,148.364
C06203=1224.268,176.326,-54.243,-177.679,5.929,148.365
C06204=1224.273,176.077,-54.220,-177.682,5.927,148.365
C06205=1224.277,175.828,-54.197,-177.684,5.926,148.365
C06206=1224.282,175.579,-54.175,-177.687,5.925,148.366
C06207=1224.286,175.330,-54.153,-177.690,5.923,148.366
C06208=1224.290,175.081,-54.130,-177.692,5.922,148.367
C06209=1224.296,174.832,-54.108,-177.695,5.920,148.367
C06210=1224.300,174.583,-54.085,-177.698,5.918,148.368
C06211=1224.305,174.335,-54.063,-177.700,5.917,148.368
C06212=1224.310,174.085,-54.041,-177.703,5.916,148.368
C06213=1224.314,173.836,-54.018,-177.705,5.915,148.369
C06214=1224.319,173.587,-53.996,-177.708,5.913,148.369
C06215=1224.324,173.338,-53.974,-177.710,5.911,148.370
C06216=1224.328,173.090,-53.951,-177.713,5.910,148.370
C06217=1224.333,172.840,-53.929,-177.715,5.908,148.371
C06218=1224.338,172.591,-53.907,-177.718,5.908,148.371
C06219=1224.342,172.343,-53.884,-177.720,5.906,148.372
C06220=1224.346,172.094,-53.862,-177.723,5.904,148.372
C06221=1224.352,171.845,-53.840,-177.725,5.903,148.372
C06222=1224.356,171.596,-53.817,-177.728,5.902,148.373
C06223=1224.360,171.347,-53.795,-177.731,5.900,148.373
C06224=1224.366,171.098,-53.773,-177.733,5.899,148.374
C06225=1224.370,170.848,-53.751,-177.736,5.897,148.374
C06226=1224.375,170.600,-53.728,-177.738,5.896,148.375
C06227=1224.379,170.351,-53.706,-177.741,5.894,148.375
C06228=1224.385,170.102,-53.684,-177.744,5.893,148.375
C06229=1224.389,169.853,-53.662,-177.746,5.892,148.376
C06230=1224.393,169.605,-53.640,-177.749,5.890,148.376
C06231=1224.398,169.355,-53.618,-177.751,5.889,148.377
C06232=1224.403,169.106,-53.595,-177.754,5.887,148.377
C06233=1224.408,168.857,-53.573,-177.757,5.886,148.378
C06234=1224.412,168.608,-53.551,-177.759,5.885,148.378
C06235=1224.417,168.359,-53.530,-177.762,5.883,148.378
C06236=1224.422,168.109,-53.507,-177.764,5.882,148.379
C06237=1224.426,167.861,-53.484,-177.767,5.881,148.379
C06238=1224.431,167.612,-53.462,-177.769,5.879,148.380
C06239=1224.435,167.363,-53.441,-177.772,5.878,148.380
C06240=1224.440,167.114,-53.419,-177.775,5.876,148.381
C06241=1224.445,166.865,-53.397,-177.777,5.875,148.381
C06242=1224.450,166.616,-53.374,-177.779,5.873,148.381
C06243=1224.454,166.367,-53.353,-177.782,5.873,148.382
C06244=1224.459,166.118,-53.331,-177.785,5.871,148.382
C06245=1224.464,165.869,-53.309,-177.787,5.869,148.383
C06246=1224.468,165.620,-53.287,-177.789,5.868,148.383
C06247=1224.473,165.371,-53.265,-177.793,5.867,148.384
C06248=1224.478,165.122,-53.244,-177.795,5.866,148.384
C06249=1224.482,164.873,-53.222,-177.797,5.864,148.385
C06250=1224.487,164.624,-53.199,-177.800,5.863,148.385
C06251=1224.492,164.375,-53.177,-177.803,5.861,148.385
C06252=1224.497,164.126,-53.156,-177.805,5.859,148.386
C06253=1224.501,163.877,-53.133,-177.808,5.859,148.386
C06254=1224.506,163.628,-53.112,-177.810,5.857,148.387
C06255=1224.510,163.379,-53.090,-177.813,5.856,148.387
C06256=1224.515,163.130,-53.068,-177.816,5.854,148.388
C06257=1224.520,162.882,-53.046,-177.818,5.853,148.388
C06258=1224.524,162.632,-53.024,-177.821,5.852,148.389
C06259=1224.529,162.384,-53.003,-177.823,5.851,148.389
C06260=1224.533,162.134,-52.981,-177.826,5.849,148.390
C06261=1224.538,161.886,-52.959,-177.828,5.847,148.390
C06262=1224.542,161.636,-52.937,-177.831,5.847,148.391
C06263=1224.547,161.387,-52.916,-177.834,5.845,148.391
C06264=1224.552,161.138,-52.894,-177.836,5.844,148.391
C06265=1224.557,160.889,-52.872,-177.839,5.842,148.392
C06266=1224.561,160.640,-52.850,-177.841,5.841,148.392
C06267=1224.566,160.391,-52.828,-177.844,5.840,148.393
C06268=1224.571,160.142,-52.807,-177.846,5.839,148.393
C06269=1224.576,159.873,-52.783,-177.849,5.837,148.394
C06270=1224.582,159.604,-52.760,-177.852,5.836,148.394
C06271=1224.586,159.335,-52.737,-177.855,5.834,148.395
C06272=1224.591,159.066,-52.713,-177.857,5.833,148.395
C06273=1224.596,158.817,-52.692,-177.860,5.831,148.396
C06274=1224.601,158.568,-52.669,-177.862,5.830,148.396
C06275=1224.606,158.319,-52.648,-177.865,5.829,148.397
C06276=1224.610,158.069,-52.626,-177.867,5.828,148.397
C06277=1224.614,157.821,-52.605,-177.870,5.826,148.397
C06278=1224.619,157.572,-52.584,-177.873,5.825,148.398
C06279=1224.624,157.322,-52.562,-177.875,5.824,148.398
C06280=1224.628,157.074,-52.541,-177.877,5.823,148.399
C06281=1224.633,156.825,-52.519,-177.881,5.821,148.399
C06282=1224.638,156.575,-52.498,-177.883,5.819,148.400
C06283=1224.643,156.326,-52.476,-177.886,5.819,148.400
C06284=1224.648,156.078,-52.454,-177.888,5.817,148.401
C06285=1224.653,155.829,-52.433,-177.891,5.816,148.401
C06286=1224.656,155.580,-52.412,-177.894,5.814,148.402
C06287=1224.661,155.331,-52.390,-177.896,5.813,148.402
C06288=1224.666,155.082,-52.369,-177.898,5.812,148.402
C06289=1224.671,154.832,-52.347,-177.901,5.811,148.403
C06290=1224.676,154.583,-52.326,-177.904,5.809,148.403
C06291=1224.681,154.334,-52.305,-177.906,5.808,148.404
C06292=1224.685,154.086,-52.283,-177.909,5.807,148.404
C06293=1224.689,153.836,-52.262,-177.911,5.806,148.405
C06294=1224.694,153.587,-52.240,-177.914,5.804,148.405
C06295=1224.699,153.338,-52.219,-177.916,5.803,148.406
C06296=1224.704,153.089,-52.197,-177.919,5.801,148.406
C06297=1224.709,152.840,-52.176,-177.922,5.801,148.407
C06298=1224.713,152.591,-52.155,-177.924,5.799,148.407
C06299=1224.718,152.342,-52.134,-177.926,5.798,148.408
C06300=1224.722,152.093,-52.112,-177.929,5.796,148.408
C06301=1224.728,151.843,-52.091,-177.932,5.795,148.409
C06302=1224.732,151.595,-52.070,-177.935,5.794,148.409
C06303=1224.737,151.346,-52.049,-177.937,5.793,148.410
C06304=1224.742,151.097,-52.028,-177.939,5.792,148.410
C06305=1224.746,150.847,-52.006,-177.942,5.790,148.411
C06306=1224.751,150.599,-51.985,-177.944,5.789,148.411
C06307=1224.756,150.350,-51.964,-177.947,5.788,148.412
C06308=1224.761,150.100,-51.943,-177.949,5.787,148.412
C06309=1224.764,149.851,-51.922,-177.952,5.785,148.412
C06310=1224.770,149.602,-51.901,-177.955,5.785,148.413
C06311=1224.774,149.353,-51.879,-177.957,5.783,148.413
C06312=1224.780,149.104,-51.858,-177.960,5.782,148.414
C06313=1224.784,148.855,-51.838,-177.963,5.780,148.414
C06314=1224.788,148.606,-51.816,-177.965,5.779,148.415
C06315=1224.794,148.357,-51.795,-177.968,5.778,148.415
C06316=1224.798,148.108,-51.774,-177.970,5.777,148.416
C06317=1224.803,147.859,-51.753,-177.973,5.775,148.416
C06318=1224.808,147.610,-51.732,-177.975,5.774,148.417
C06319=1224.812,147.361,-51.711,-177.978,5.773,148.417
C06320=1224.817,147.112,-51.689,-177.981,5.772,148.418
C06321=1224.821,146.863,-51.669,-177.983,5.771,148.418
C06322=1224.826,146.613,-51.648,-177.986,5.769,148.419
C06323=1224.831,146.365,-51.626,-177.988,5.768,148.419
C06324=1224.836,146.116,-51.606,-177.991,5.767,148.420
C06325=1224.841,145.866,-51.585,-177.993,5.766,148.420
C06326=1224.846,145.617,-51.564,-177.996,5.764,148.420
C06327=1224.849,145.368,-51.543,-177.998,5.764,148.421
C06328=1224.855,145.119,-51.522,-178.001,5.762,148.421
C06329=1224.859,144.870,-51.501,-178.004,5.761,148.422
C06330=1224.864,144.621,-51.480,-178.006,5.760,148.423
C06331=1224.868,144.372,-51.459,-178.009,5.758,148.423
C06332=1224.874,144.123,-51.438,-178.011,5.758,148.424
C06333=1224.878,143.874,-51.418,-178.014,5.756,148.424
C06334=1224.883,143.625,-51.397,-178.016,5.755,148.425
C06335=1224.888,143.375,-51.376,-178.019,5.753,148.425
C06336=1224.892,143.126,-51.355,-178.022,5.753,148.426
C06337=1224.897,142.877,-51.334,-178.024,5.751,148.426
C06338=1224.902,142.628,-51.313,-178.027,5.750,148.427
C06339=1224.907,142.379,-51.292,-178.029,5.749,148.427
C06340=1224.911,142.130,-51.272,-178.032,5.748,148.427
C06341=1224.916,141.881,-51.251,-178.034,5.747,148.428
C06342=1224.921,141.632,-51.230,-178.037,5.745,148.428
C06343=1224.926,141.383,-51.209,-178.040,5.744,148.429
C06344=1224.930,141.134,-51.189,-178.042,5.743,148.429
C06345=1224.936,140.885,-51.168,-178.045,5.742,148.430
C06346=1224.940,140.636,-51.148,-178.047,5.741,148.430
C06347=1224.944,140.387,-51.127,-178.050,5.740,148.431
C06348=1224.949,140.137,-51.105,-178.052,5.739,148.431
C06349=1224.953,139.888,-51.085,-178.055,5.737,148.432
C06350=1224.958,139.639,-51.064,-178.057,5.736,148.432
C06351=1224.963,139.390,-51.044,-178.060,5.735,148.433
C06352=1224.968,139.141,-51.023,-178.063,5.734,148.433
C06353=1224.972,138.892,-51.002,-178.065,5.733,148.434
C06354=1224.977,138.643,-50.982,-178.068,5.731,148.434
C06355=1224.982,138.394,-50.961,-178.070,5.730,148.435
C06356=1224.987,138.144,-50.941,-178.073,5.730,148.435
C06357=1224.992,137.895,-50.920,-178.075,5.728,148.436
C06358=1224.996,137.646,-50.900,-178.078,5.727,148.436
C06359=1225.001,137.397,-50.880,-178.081,5.725,148.437
C06360=1225.006,137.148,-50.859,-178.083,5.725,148.437
C06361=1225.010,136.899,-50.838,-178.085,5.724,148.438
C06362=1225.016,136.650,-50.817,-178.088,5.722,148.438
C06363=1225.020,136.401,-50.797,-178.091,5.721,148.439
C06364=1225.024,136.152,-50.777,-178.093,5.719,148.439
C06365=1225.030,135.902,-50.756,-178.096,5.719,148.440
C06366=1225.034,135.653,-50.735,-178.098,5.718,148.440
C06367=1225.039,135.404,-50.716,-178.101,5.716,148.441
C06368=1225.044,135.155,-50.695,-178.103,5.715,148.441
C06369=1225.048,134.906,-50.674,-178.106,5.714,148.442
C06370=1225.053,134.657,-50.654,-178.109,5.713,148.442
C06371=1225.059,134.408,-50.633,-178.111,5.712,148.443
C06372=1225.063,134.159,-50.613,-178.114,5.711,148.443
C06373=1225.067,133.890,-50.591,-178.116,5.710,148.444
C06374=1225.073,133.621,-50.569,-178.120,5.708,148.445
C06375=1225.078,133.353,-50.547,-178.122,5.707,148.445
C06376=1225.084,133.084,-50.525,-178.125,5.706,148.446
C06377=1225.088,132.835,-50.505,-178.128,5.705,148.446
C06378=1225.093,132.586,-50.485,-178.130,5.704,148.447
C06379=1225.097,132.337,-50.465,-178.133,5.703,148.447
C06380=1225.102,132.087,-50.444,-178.135,5.702,148.448
C06381=1225.107,131.838,-50.424,-178.138,5.700,148.448
C06382=1225.112,131.589,-50.404,-178.140,5.700,148.449
C06383=1225.116,131.340,-50.383,-178.143,5.698,148.449
C06384=1225.121,131.092,-50.363,-178.145,5.697,148.450
C06385=1225.127,130.842,-50.343,-178.148,5.696,148.450
C06386=1225.131,130.593,-50.323,-178.151,5.695,148.451
C06387=1225.135,130.344,-50.302,-178.153,5.694,148.451
C06388=1225.140,130.094,-50.283,-178.155,5.693,148.452
C06389=1225.145,129.845,-50.262,-178.159,5.692,148.452
C06390=1225.150,129.596,-50.242,-178.161,5.691,148.453
C06391=1225.155,129.347,-50.222,-178.163,5.690,148.453
C06392=1225.159,129.098,-50.201,-178.166,5.688,148.454
C06393=1225.164,128.849,-50.182,-178.169,5.688,148.454
C06394=1225.169,128.600,-50.161,-178.171,5.687,148.455
C06395=1225.173,128.351,-50.141,-178.174,5.685,148.455
C06396=1225.179,128.101,-50.121,-178.176,5.684,148.456
C06397=1225.183,127.852,-50.100,-178.179,5.683,148.456
C06398=1225.188,127.602,-50.081,-178.181,5.682,148.457
C06399=1225.193,127.354,-50.061,-178.184,5.681,148.457
C06400=1225.198,127.105,-50.041,-178.187,5.679,148.458
C06401=1225.202,126.856,-50.021,-178.189,5.679,148.458
C06402=1225.207,126.606,-50.001,-178.191,5.678,148.459
C06403=1225.211,126.357,-49.981,-178.194,5.676,148.460
C06404=1225.216,126.108,-49.961,-178.197,5.675,148.460
C06405=1225.221,125.859,-49.941,-178.199,5.675,148.461
C06406=1225.227,125.610,-49.921,-178.202,5.673,148.461
C06407=1225.231,125.361,-49.900,-178.204,5.672,148.462
C06408=1225.236,125.111,-49.881,-178.207,5.672,148.462
C06409=1225.240,124.862,-49.860,-178.210,5.670,148.463
C06410=1225.246,124.613,-49.841,-178.212,5.669,148.463
C06411=1225.250,124.364,-49.821,-178.214,5.668,148.464
C06412=1225.255,124.115,-49.801,-178.217,5.668,148.464
C06413=1225.259,123.866,-49.781,-178.220,5.666,148.465
C06414=1225.264,123.616,-49.761,-178.222,5.665,148.465
C06415=1225.269,123.367,-49.742,-178.224,5.664,148.466
C06416=1225.274,123.118,-49.721,-178.228,5.663,148.466
C06417=1225.278,122.869,-49.702,-178.230,5.662,148.467
C06418=1225.283,122.620,-49.681,-178.232,5.661,148.467
C06419=1225.288,122.371,-49.662,-178.236,5.660,148.468
C06420=1225.293,122.121,-49.642,-178.238,5.659,148.468
C06421=1225.297,121.872,-49.622,-178.240,5.658,148.469
C06422=1225.302,121.623,-49.602,-178.243,5.656,148.469
C06423=1225.307,121.374,-49.583,-178.246,5.656,148.470
C06424=1225.312,121.125,-49.563,-178.248,5.655,148.470
C06425=1225.317,120.875,-49.543,-178.251,5.653,148.471
C06426=1225.321,120.626,-49.523,-178.253,5.652,148.472
C06427=1225.327,120.377,-49.504,-178.256,5.652,148.472
C06428=1225.331,120.128,-49.484,-178.258,5.651,148.473
C06429=1225.335,119.879,-49.465,-178.261,5.649,148.473
C06430=1225.340,119.630,-49.445,-178.263,5.649,148.474
C06431=1225.345,119.381,-49.425,-178.266,5.648,148.474
C06432=1225.350,119.131,-49.405,-178.269,5.646,148.475
C06433=1225.354,118.882,-49.386,-178.271,5.645,148.475
C06434=1225.360,118.633,-49.366,-178.273,5.645,148.476
C06435=1225.365,118.383,-49.347,-178.276,5.644,148.477
C06436=1225.369,118.135,-49.326,-178.279,5.642,148.477
C06437=1225.374,117.886,-49.307,-178.281,5.642,148.478
C06438=1225.379,117.636,-49.288,-178.284,5.641,148.478
C06439=1225.383,117.387,-49.268,-178.287,5.639,148.479
C06440=1225.388,117.138,-49.249,-178.289,5.638,148.479
C06441=1225.393,116.889,-49.229,-178.291,5.638,148.480
C06442=1225.398,116.639,-49.209,-178.294,5.637,148.480
C06443=1225.403,116.391,-49.190,-178.297,5.635,148.481
C06444=1225.408,116.141,-49.170,-178.299,5.634,148.481
C06445=1225.412,115.892,-49.151,-178.301,5.634,148.482
C06446=1225.417,115.643,-49.132,-178.305,5.632,148.482
C06447=1225.422,115.393,-49.112,-178.307,5.631,148.483
C06448=1225.427,115.144,-49.093,-178.309,5.630,148.483
C06449=1225.432,114.895,-49.073,-178.312,5.630,148.484
C06450=1225.436,114.646,-49.053,-178.315,5.628,148.484
C06451=1225.441,114.397,-49.034,-178.317,5.627,148.485
C06452=1225.446,114.148,-49.015,-178.319,5.626,148.486
C06453=1225.450,113.898,-48.995,-178.322,5.626,148.486
C06454=1225.456,113.649,-48.976,-178.325,5.624,148.487
C06455=1225.460,113.400,-48.957,-178.327,5.623,148.487
C06456=1225.465,113.151,-48.937,-178.330,5.623,148.488
C06457=1225.470,112.902,-48.918,-178.332,5.622,148.488
C06458=1225.475,112.652,-48.898,-178.335,5.620,148.489
C06459=1225.479,112.404,-48.879,-178.338,5.620,148.490
C06460=1225.484,112.154,-48.860,-178.340,5.619,148.490
C06461=1225.489,111.905,-48.840,-178.343,5.618,148.491
C06462=1225.494,111.656,-48.821,-178.345,5.616,148.491
C06463=1225.499,111.407,-48.802,-178.348,5.616,148.492
C06464=1225.503,111.157,-48.782,-178.350,5.615,148.492
C06465=1225.508,110.908,-48.763,-178.353,5.614,148.493
C06466=1225.513,110.659,-48.744,-178.356,5.613,148.493
C06467=1225.518,110.409,-48.725,-178.358,5.612,148.494
C06468=1225.523,110.160,-48.706,-178.360,5.611,148.494
C06469=1225.527,109.911,-48.687,-178.363,5.611,148.495
C06470=1225.532,109.662,-48.667,-178.366,5.609,148.495
C06471=1225.537,109.413,-48.648,-178.368,5.608,148.496
C06472=1225.541,109.163,-48.629,-178.371,5.608,148.497
C06473=1225.546,108.914,-48.609,-178.373,5.607,148.497
C06474=1225.551,108.665,-48.590,-178.376,5.605,148.498
C06475=1225.556,108.416,-48.571,-178.378,5.604,148.498
C06476=1225.561,108.166,-48.552,-178.381,5.604,148.499
C06477=1225.566,107.898,-48.531,-178.384,5.602,148.499
C06478=1225.571,107.630,-48.510,-178.387,5.602,148.500
C06479=1225.576,107.361,-48.491,-178.389,5.601,148.501
C06480=1225.581,107.093,-48.470,-178.392,5.599,148.501
C06481=1225.587,106.844,-48.450,-178.395,5.599,148.502
C06482=1225.591,106.594,-48.431,-178.397,5.598,148.502
C06483=1225.596,106.345,-48.413,-178.399,5.597,148.503
C06484=1225.601,106.095,-48.393,-178.403,5.596,148.503
C06485=1225.606,105.847,-48.374,-178.405,5.595,148.504
C06486=1225.610,105.597,-48.355,-178.407,5.594,148.504
C06487=1225.615,105.348,-48.337,-178.410,5.593,148.505
C06488=1225.620,105.099,-48.317,-178.413,5.593,148.506
C06489=1225.625,104.850,-48.298,-178.415,5.591,148.506
C06490=1225.629,104.600,-48.279,-178.418,5.590,148.507
C06491=1225.635,104.351,-48.260,-178.420,5.589,148.507
C06492=1225.640,104.102,-48.242,-178.423,5.589,148.508
C06493=1225.644,103.853,-48.222,-178.426,5.587,148.509
C06494=1225.649,103.604,-48.204,-178.428,5.586,148.509
C06495=1225.654,103.354,-48.184,-178.431,5.586,148.510
C06496=1225.659,103.106,-48.166,-178.433,5.585,148.510
C06497=1225.664,102.855,-48.147,-178.435,5.584,148.511
C06498=1225.668,102.607,-48.128,-178.439,5.583,148.511
C06499=1225.673,102.357,-48.108,-178.441,5.582,148.512
C06500=1225.678,102.108,-48.090,-178.443,5.581,148.512
C06501=1225.683,101.859,-48.071,-178.446,5.581,148.513
C06502=1225.688,101.609,-48.053,-178.448,5.580,148.514
C06503=1225.692,101.361,-48.034,-178.451,5.578,148.514
C06504=1225.697,101.111,-48.014,-178.454,5.578,148.515
C06505=1225.702,100.862,-47.996,-178.456,5.577,148.515
C06506=1225.707,100.612,-47.977,-178.459,5.576,148.516
C06507=1225.712,100.363,-47.959,-178.461,5.575,148.516
C06508=1225.717,100.114,-47.939,-178.464,5.575,148.517
C06509=1225.721,99.864,-47.921,-178.466,5.573,148.517
C06510=1225.726,99.616,-47.902,-178.469,5.572,148.518
C06511=1225.731,99.366,-47.884,-178.472,5.572,148.519
C06512=1225.735,99.117,-47.865,-178.474,5.571,148.519
C06513=1225.741,98.868,-47.846,-178.476,5.570,148.520
C06514=1225.745,98.618,-47.827,-178.480,5.569,148.520
C06515=1225.750,98.369,-47.809,-178.482,5.568,148.521
C06516=1225.755,98.120,-47.790,-178.484,5.567,148.522
C06517=1225.760,97.871,-47.771,-178.487,5.567,148.522
C06518=1225.765,97.622,-47.752,-178.489,5.566,148.523
C06519=1225.770,97.372,-47.734,-178.492,5.565,148.523
C06520=1225.774,97.123,-47.715,-178.495,5.564,148.524
C06521=1225.780,96.874,-47.697,-178.497,5.563,148.524
C06522=1225.784,96.625,-47.678,-178.500,5.562,148.525
C06523=1225.789,96.375,-47.659,-178.502,5.562,148.526
C06524=1225.794,96.126,-47.641,-178.504,5.561,148.526
C06525=1225.799,95.877,-47.622,-178.507,5.560,148.527
C06526=1225.803,95.627,-47.604,-178.510,5.559,148.527
C06527=1225.808,95.379,-47.585,-178.512,5.558,148.528
C06528=1225.813,95.129,-47.567,-178.515,5.557,148.528
C06529=1225.818,94.879,-47.548,-178.518,5.556,148.529
C06530=1225.823,94.631,-47.529,-178.520,5.556,148.530
C06531=1225.828,94.381,-47.511,-178.522,5.555,148.530
C06532=1225.832,94.132,-47.493,-178.526,5.553,148.531
C06533=1225.837,93.883,-47.474,-178.528,5.553,148.531
C06534=1225.842,93.634,-47.455,-178.530,5.552,148.532
C06535=1225.847,93.384,-47.437,-178.533,5.551,148.532
C06536=1225.852,93.134,-47.419,-178.536,5.551,148.533
C06537=1225.856,92.886,-47.400,-178.538,5.550,148.534
C06538=1225.862,92.636,-47.382,-178.540,5.549,148.534
C06539=1225.866,92.387,-47.363,-178.543,5.548,148.535
C06540=1225.871,92.138,-47.345,-178.546,5.547,148.535
C06541=1225.876,91.889,-47.327,-178.548,5.546,148.536
C06542=1225.881,91.639,-47.308,-178.551,5.545,148.537
C06543=1225.886,91.389,-47.290,-178.553,5.545,148.537
C06544=1225.890,91.141,-47.271,-178.556,5.544,148.538
C06545=1225.895,90.892,-47.253,-178.558,5.543,148.538
C06546=1225.900,90.643,-47.235,-178.561,5.542,148.539
C06547=1225.905,90.392,-47.216,-178.563,5.541,148.539
C06548=1225.910,90.143,-47.198,-178.566,5.540,148.540
C06549=1225.915,89.895,-47.180,-178.569,5.540,148.541
C06550=1225.920,89.645,-47.162,-178.571,5.539,148.541
C06551=1225.924,89.396,-47.143,-178.573,5.538,148.542
C06552=1225.929,89.146,-47.125,-178.576,5.538,148.542
C06553=1225.935,88.897,-47.107,-178.579,5.537,148.543
C06554=1225.939,88.648,-47.089,-178.581,5.535,148.543
C06555=1225.944,88.399,-47.071,-178.584,5.535,148.544
C06556=1225.948,88.149,-47.052,-178.587,5.534,148.545
C06557=1225.953,87.900,-47.034,-178.589,5.533,148.545
C06558=1225.958,87.651,-47.016,-178.591,5.532,148.546
C06559=1225.963,87.402,-46.998,-178.594,5.532,148.546
C06560=1225.968,87.153,-46.980,-178.597,5.531,148.547
C06561=1225.973,86.902,-46.961,-178.599,5.531,148.548
C06562=1225.978,86.653,-46.943,-178.602,5.529,148.548
C06563=1225.983,86.404,-46.925,-178.605,5.528,148.549
C06564=1225.988,86.155,-46.907,-178.607,5.528,148.549
C06565=1225.993,85.906,-46.889,-178.609,5.527,148.550
C06566=1225.997,85.656,-46.871,-178.612,5.526,148.551
C06567=1226.002,85.407,-46.853,-178.615,5.526,148.551
C06568=1226.007,85.157,-46.835,-178.617,5.525,148.552
C06569=1226.012,84.908,-46.817,-178.619,5.524,148.552
C06570=1226.017,84.659,-46.799,-178.622,5.523,148.553
C06571=1226.022,84.410,-46.781,-178.625,5.522,148.554
C06572=1226.026,84.161,-46.763,-178.628,5.521,148.554
C06573=1226.031,83.911,-46.744,-178.630,5.520,148.555
C06574=1226.036,83.662,-46.726,-178.633,5.520,148.555
C06575=1226.041,83.413,-46.708,-178.635,5.519,148.556
C06576=1226.046,83.163,-46.690,-178.638,5.519,148.557
C06577=1226.050,82.914,-46.672,-178.640,5.518,148.557
C06578=1226.055,82.665,-46.654,-178.643,5.517,148.558
C06579=1226.060,82.416,-46.636,-178.645,5.517,148.558
C06580=1226.065,82.167,-46.618,-178.648,5.516,148.559
C06581=1226.070,81.898,-46.599,-178.651,5.515,148.560
C06582=1226.076,81.630,-46.580,-178.653,5.514,148.560
C06583=1226.081,81.361,-46.560,-178.656,5.513,148.561
C06584=1226.087,81.093,-46.541,-178.658,5.512,148.561
C06585=1226.091,80.844,-46.523,-178.662,5.511,148.562
C06586=1226.096,80.594,-46.505,-178.664,5.510,148.563
C06587=1226.100,80.344,-46.488,-178.667,5.510,148.563
C06588=1226.105,80.095,-46.470,-178.669,5.509,148.564
C06589=1226.110,79.846,-46.452,-178.672,5.508,148.564
C06590=1226.115,79.597,-46.434,-178.674,5.508,148.565
C06591=1226.120,79.347,-46.416,-178.677,5.507,148.566
C06592=1226.125,79.098,-46.398,-178.679,5.506,148.566
C06593=1226.130,78.849,-46.381,-178.682,5.506,148.567
C06594=1226.135,78.599,-46.363,-178.684,5.505,148.568
C06595=1226.140,78.350,-46.345,-178.687,5.504,148.568
C06596=1226.145,78.101,-46.327,-178.689,5.504,148.569
C06597=1226.150,77.851,-46.310,-178.692,5.503,148.569
C06598=1226.154,77.602,-46.292,-178.695,5.501,148.570
C06599=1226.159,77.353,-46.274,-178.697,5.501,148.571
C06600=1226.164,77.104,-46.256,-178.700,5.500,148.571
C06601=1226.169,76.854,-46.239,-178.702,5.499,148.572
C06602=1226.174,76.605,-46.221,-178.705,5.499,148.572
C06603=1226.179,76.356,-46.203,-178.707,5.498,148.573
C06604=1226.184,76.106,-46.186,-178.710,5.498,148.574
C06605=1226.188,75.857,-46.168,-178.712,5.497,148.574
C06606=1226.193,75.608,-46.150,-178.715,5.496,148.575
C06607=1226.198,75.359,-46.132,-178.717,5.495,148.575
C06608=1226.203,75.109,-46.115,-178.720,5.495,148.576
C06609=1226.208,74.860,-46.097,-178.723,5.494,148.577
C06610=1226.213,74.610,-46.080,-178.725,5.493,148.577
C06611=1226.218,74.361,-46.063,-178.727,5.493,148.578
C06612=1226.223,74.112,-46.045,-178.730,5.492,148.578
C06613=1226.228,73.862,-46.027,-178.733,5.492,148.579
C06614=1226.233,73.613,-46.009,-178.735,5.491,148.580
C06615=1226.237,73.364,-45.992,-178.738,5.490,148.580
C06616=1226.242,73.114,-45.975,-178.741,5.489,148.581
C06617=1226.247,72.865,-45.957,-178.743,5.488,148.581
C06618=1226.252,72.615,-45.939,-178.746,5.487,148.582
C06619=1226.257,72.367,-45.922,-178.748,5.487,148.583
C06620=1226.262,72.117,-45.905,-178.751,5.486,148.583
C06621=1226.267,71.868,-45.887,-178.753,5.485,148.584
C06622=1226.272,71.618,-45.869,-178.756,5.485,148.585
C06623=1226.276,71.369,-45.852,-178.759,5.484,148.585
C06624=1226.281,71.120,-45.834,-178.761,5.483,148.586
C06625=1226.286,70.870,-45.817,-178.763,5.483,148.586
C06626=1226.291,70.621,-45.799,-178.766,5.482,148.587
C06627=1226.296,70.371,-45.782,-178.769,5.482,148.588
C06628=1226.300,70.122,-45.764,-178.771,5.481,148.588
C06629=1226.306,69.872,-45.747,-178.773,5.480,148.589
C06630=1226.310,69.623,-45.730,-178.776,5.479,148.589
C06631=1226.316,69.374,-45.713,-178.779,5.479,148.590
C06632=1226.321,69.125,-45.695,-178.781,5.478,148.591
C06633=1226.325,68.876,-45.678,-178.784,5.478,148.591
C06634=1226.330,68.626,-45.661,-178.786,5.477,148.592
C06635=1226.335,68.377,-45.643,-178.789,5.476,148.592
C06636=1226.340,68.127,-45.626,-178.791,5.476,148.593
C06637=1226.345,67.878,-45.608,-178.794,5.475,148.594
C06638=1226.350,67.628,-45.591,-178.797,5.474,148.594
C06639=1226.354,67.379,-45.574,-178.799,5.473,148.595
C06640=1226.359,67.130,-45.556,-178.801,5.473,148.596
C06641=1226.364,66.881,-45.540,-178.804,5.472,148.596
C06642=1226.369,66.632,-45.522,-178.807,5.472,148.597
C06643=1226.374,66.382,-45.505,-178.809,5.471,148.598
C06644=1226.379,66.132,-45.488,-178.811,5.470,148.598
C06645=1226.384,65.883,-45.470,-178.814,5.470,148.599
C06646=1226.388,65.634,-45.453,-178.817,5.469,148.599
C06647=1226.394,65.384,-45.436,-178.819,5.468,148.600
C06648=1226.399,65.135,-45.418,-178.822,5.468,148.601
C06649=1226.403,64.886,-45.402,-178.825,5.467,148.601
C06650=1226.409,64.636,-45.385,-178.827,5.466,148.602
C06651=1226.413,64.387,-45.367,-178.829,5.466,148.602
C06652=1226.418,64.138,-45.350,-178.832,5.465,148.603
C06653=1226.423,63.888,-45.333,-178.835,5.465,148.604
C06654=1226.428,63.639,-45.316,-178.837,5.464,148.604
C06655=1226.433,63.390,-45.299,-178.839,5.463,148.605
C06656=1226.438,63.140,-45.282,-178.842,5.463,148.605
C06657=1226.442,62.891,-45.265,-178.845,5.462,148.606
C06658=1226.447,62.641,-45.248,-178.847,5.461,148.607
C06659=1226.452,62.392,-45.230,-178.850,5.461,148.607
C06660=1226.457,62.143,-45.213,-178.852,5.460,148.608
C06661=1226.462,61.894,-45.197,-178.855,5.459,148.609
C06662=1226.467,61.644,-45.180,-178.857,5.459,148.609
C06663=1226.472,61.394,-45.163,-178.860,5.458,148.610
C06664=1226.477,61.145,-45.145,-178.863,5.458,148.611
C06665=1226.482,60.896,-45.129,-178.865,5.457,148.611
C06666=1226.487,60.647,-45.111,-178.868,5.456,148.612
C06667=1226.491,60.397,-45.095,-178.870,5.455,148.612
C06668=1226.497,60.147,-45.077,-178.873,5.455,148.613
C06669=1226.502,59.898,-45.061,-178.875,5.454,148.614
C06670=1226.507,59.649,-45.044,-178.878,5.454,148.614
C06671=1226.511,59.400,-45.026,-178.880,5.453,148.615
C06672=1226.516,59.150,-45.009,-178.883,5.453,148.616
C06673=1226.521,58.901,-44.993,-178.885,5.452,148.616
C06674=1226.526,58.652,-44.976,-178.888,5.451,148.617
C06675=1226.531,58.402,-44.959,-178.891,5.451,148.617
C06676=1226.536,58.152,-44.942,-178.893,5.450,148.618
C06677=1226.541,57.903,-44.925,-178.896,5.449,148.619
C06678=1226.546,57.654,-44.909,-178.898,5.449,148.619
C06679=1226.550,57.404,-44.892,-178.901,5.448,148.620
C06680=1226.556,57.155,-44.875,-178.903,5.447,148.621
C06681=1226.561,56.906,-44.858,-178.906,5.447,148.621
C06682=1226.566,56.656,-44.841,-178.908,5.446,148.622
C06683=1226.570,56.407,-44.825,-178.911,5.446,148.623
C06684=1226.575,56.158,-44.808,-178.914,5.445,148.623
C06685=1226.581,55.889,-44.790,-178.916,5.444,148.624
C06686=1226.586,55.621,-44.772,-178.919,5.444,148.625
C06687=1226.591,55.352,-44.753,-178.922,5.443,148.625
C06688=1226.597,55.084,-44.735,-178.924,5.443,148.626
C06689=1226.601,54.835,-44.719,-178.927,5.442,148.627
C06690=1226.606,54.585,-44.701,-178.930,5.442,148.627
C06691=1226.611,54.336,-44.685,-178.932,5.441,148.628
C06692=1226.616,54.087,-44.668,-178.935,5.440,148.629
C06693=1226.621,53.837,-44.651,-178.937,5.440,148.629
C06694=1226.626,53.587,-44.635,-178.940,5.439,148.630
C06695=1226.631,53.338,-44.619,-178.942,5.438,148.630
C06696=1226.636,53.088,-44.602,-178.945,5.438,148.631
C06697=1226.641,52.839,-44.585,-178.947,5.437,148.632
C06698=1226.646,52.590,-44.569,-178.950,5.437,148.632
C06699=1226.650,52.341,-44.552,-178.953,5.436,148.633
C06700=1226.655,52.091,-44.535,-178.955,5.435,148.633
C06701=1226.661,51.842,-44.518,-178.958,5.435,148.634
C06702=1226.665,51.592,-44.502,-178.960,5.434,148.635
C06703=1226.670,51.343,-44.486,-178.963,5.433,148.635
C06704=1226.676,51.093,-44.469,-178.965,5.434,148.636
C06705=1226.680,50.844,-44.452,-178.968,5.433,148.637
C06706=1226.685,50.595,-44.436,-178.970,5.433,148.637
C06707=1226.690,50.346,-44.419,-178.972,5.432,148.638
C06708=1226.695,50.096,-44.402,-178.975,5.431,148.639
C06709=1226.700,49.846,-44.386,-178.978,5.431,148.639
C06710=1226.705,49.597,-44.370,-178.980,5.430,148.640
C06711=1226.710,49.348,-44.353,-178.983,5.429,148.641
C06712=1226.714,49.099,-44.337,-178.985,5.429,148.641
C06713=1226.720,48.849,-44.320,-178.988,5.428,148.642
C06714=1226.725,48.599,-44.304,-178.991,5.428,148.643
C06715=1226.729,48.350,-44.287,-178.993,5.427,148.643
C06716=1226.734,48.101,-44.271,-178.996,5.426,148.644
C06717=1226.739,47.852,-44.254,-178.998,5.426,148.644
C06718=1226.744,47.601,-44.238,-179.001,5.425,148.645
C06719=1226.750,47.352,-44.221,-179.003,5.425,148.646
C06720=1226.754,47.103,-44.205,-179.006,5.425,148.646
C06721=1226.759,46.854,-44.189,-179.008,5.424,148.647
C06722=1226.764,46.604,-44.173,-179.011,5.424,148.648
C06723=1226.769,46.355,-44.156,-179.013,5.423,148.648
C06724=1226.774,46.105,-44.140,-179.016,5.422,148.649
C06725=1226.778,45.856,-44.124,-179.018,5.422,148.650
C06726=1226.783,45.607,-44.107,-179.021,5.421,148.650
C06727=1226.789,45.356,-44.091,-179.023,5.420,148.651
C06728=1226.794,45.108,-44.074,-179.026,5.420,148.652
C06729=1226.798,44.858,-44.058,-179.029,5.419,148.652
C06730=1226.804,44.609,-44.042,-179.031,5.419,148.653
C06731=1226.808,44.359,-44.026,-179.033,5.419,148.654
C06732=1226.813,44.111,-44.009,-179.036,5.418,148.654
C06733=1226.818,43.860,-43.993,-179.038,5.418,148.655
C06734=1226.823,43.612,-43.977,-179.041,5.417,148.655
C06735=1226.828,43.362,-43.961,-179.044,5.416,148.656
C06736=1226.833,43.113,-43.945,-179.046,5.416,148.657
C06737=1226.838,42.863,-43.929,-179.049,5.415,148.657
C06738=1226.843,42.614,-43.912,-179.051,5.415,148.658
C06739=1226.848,42.364,-43.895,-179.054,5.414,148.659
C06740=1226.854,42.115,-43.880,-179.057,5.414,148.659
C06741=1226.858,41.865,-43.863,-179.059,5.413,148.660
C06742=1226.863,41.616,-43.847,-179.061,5.413,148.661
C06743=1226.868,41.366,-43.831,-179.064,5.412,148.661
C06744=1226.873,41.117,-43.815,-179.066,5.412,148.662
C06745=1226.878,40.867,-43.798,-179.069,5.411,148.663
C06746=1226.883,40.618,-43.783,-179.072,5.411,148.663
C06747=1226.888,40.369,-43.766,-179.074,5.410,148.664
C06748=1226.893,40.119,-43.751,-179.077,5.410,148.665
C06749=1226.898,39.870,-43.734,-179.079,5.409,148.665
C06750=1226.903,39.620,-43.718,-179.082,5.409,148.666
C06751=1226.907,39.371,-43.702,-179.084,5.409,148.667
C06752=1226.913,39.121,-43.686,-179.087,5.408,148.667
C06753=1226.918,38.871,-43.670,-179.089,5.407,148.668
C06754=1226.923,38.622,-43.654,-179.092,5.407,148.668
C06755=1226.927,38.373,-43.639,-179.094,5.406,148.669
C06756=1226.932,38.124,-43.622,-179.097,5.406,148.670
C06757=1226.937,37.874,-43.607,-179.099,5.405,148.670
C06758=1226.942,37.625,-43.590,-179.102,5.405,148.671
C06759=1226.947,37.376,-43.574,-179.105,5.404,148.672
C06760=1226.952,37.125,-43.558,-179.107,5.404,148.672
C06761=1226.957,36.877,-43.542,-179.109,5.404,148.673
C06762=1226.962,36.627,-43.526,-179.112,5.403,148.674
C06763=1226.967,36.377,-43.510,-179.115,5.403,148.674
C06764=1226.972,36.128,-43.494,-179.117,5.402,148.675
C06765=1226.977,35.878,-43.478,-179.120,5.401,148.676
C06766=1226.982,35.629,-43.463,-179.122,5.401,148.676
C06767=1226.987,35.380,-43.447,-179.125,5.400,148.677
C06768=1226.991,35.130,-43.431,-179.127,5.400,148.678
C06769=1226.997,34.881,-43.415,-179.130,5.400,148.678
C06770=1227.001,34.631,-43.399,-179.132,5.399,148.679
C06771=1227.007,34.382,-43.383,-179.135,5.399,148.680
C06772=1227.012,34.133,-43.368,-179.137,5.398,148.680
C06773=1227.017,33.883,-43.351,-179.140,5.397,148.681
C06774=1227.021,33.634,-43.336,-179.143,5.397,148.682
C06775=1227.026,33.384,-43.320,-179.145,5.397,148.682
C06776=1227.031,33.135,-43.304,-179.147,5.397,148.683
C06777=1227.036,32.886,-43.288,-179.150,5.396,148.683
C06778=1227.041,32.636,-43.272,-179.152,5.395,148.684
C06779=1227.047,32.386,-43.257,-179.155,5.395,148.685
C06780=1227.051,32.137,-43.242,-179.158,5.394,148.685
C06781=1227.056,31.887,-43.226,-179.160,5.394,148.686
C06782=1227.061,31.638,-43.209,-179.162,5.394,148.687
C06783=1227.067,31.389,-43.194,-179.165,5.393,148.688
C06784=1227.071,31.139,-43.178,-179.168,5.393,148.688
C06785=1227.076,30.890,-43.163,-179.170,5.392,148.689
C06786=1227.081,30.640,-43.147,-179.173,5.392,148.690
C06787=1227.086,30.391,-43.130,-179.175,5.391,148.690
C06788=1227.091,30.141,-43.115,-179.178,5.390,148.691
C06789=1227.096,29.873,-43.098,-179.181,5.390,148.692
C06790=1227.102,29.604,-43.082,-179.183,5.389,148.692
C06791=1227.107,29.335,-43.065,-179.186,5.389,148.693
C06792=1227.112,29.066,-43.048,-179.189,5.388,148.694
C06793=1227.118,28.817,-43.032,-179.191,5.389,148.694
C06794=1227.122,28.568,-43.017,-179.193,5.388,148.695
C06795=1227.127,28.318,-43.001,-179.196,5.387,148.696
C06796=1227.133,28.068,-42.986,-179.199,5.387,148.696
C06797=1227.137,27.820,-42.970,-179.201,5.386,148.697
C06798=1227.142,27.571,-42.954,-179.204,5.386,148.698
C06799=1227.147,27.321,-42.938,-179.206,5.386,148.698
C06800=1227.153,27.071,-42.923,-179.209,5.386,148.699
C06801=1227.157,26.822,-42.908,-179.211,5.385,148.700
C06802=1227.162,26.572,-42.892,-179.214,5.384,148.700
C06803=1227.167,26.323,-42.876,-179.217,5.384,148.701
C06804=1227.172,26.073,-42.861,-179.219,5.383,148.702
C06805=1227.177,25.824,-42.846,-179.221,5.384,148.702
C06806=1227.182,25.574,-42.830,-179.224,5.383,148.703
C06807=1227.187,25.325,-42.815,-179.226,5.382,148.704
C06808=1227.192,25.075,-42.799,-179.229,5.382,148.704
C06809=1227.198,24.826,-42.784,-179.231,5.381,148.705
C06810=1227.202,24.576,-42.768,-179.234,5.381,148.706
C06811=1227.207,24.327,-42.753,-179.236,5.381,148.706
C06812=1227.212,24.078,-42.738,-179.239,5.380,148.707
C06813=1227.217,23.828,-42.722,-179.241,5.380,148.708
C06814=1227.222,23.579,-42.706,-179.244,5.379,148.708
C06815=1227.227,23.329,-42.691,-179.247,5.379,148.709
C06816=1227.232,23.080,-42.675,-179.249,5.378,148.710
C06817=1227.237,22.830,-42.661,-179.251,5.378,148.710
C06818=1227.242,22.581,-42.646,-179.254,5.378,148.711
C06819=1227.247,22.331,-42.630,-179.257,5.377,148.712
C06820=1227.252,22.081,-42.615,-179.259,5.377,148.712
C06821=1227.257,21.832,-42.599,-179.262,5.376,148.713
C06822=1227.262,21.583,-42.584,-179.264,5.376,148.714
C06823=1227.267,21.334,-42.569,-179.267,5.376,148.714
C06824=1227.271,21.084,-42.553,-179.269,5.375,148.715
C06825=1227.277,20.834,-42.538,-179.272,5.375,148.716
C06826=1227.282,20.584,-42.523,-179.275,5.374,148.717
C06827=1227.287,20.335,-42.508,-179.276,5.374,148.717
C06828=1227.292,20.086,-42.492,-179.279,5.374,148.718
C06829=1227.297,19.837,-42.477,-179.282,5.373,148.718
C06830=1227.302,19.587,-42.461,-179.284,5.373,148.719
C06831=1227.307,19.337,-42.447,-179.287,5.372,148.720
C06832=1227.312,19.088,-42.431,-179.289,5.372,148.720
C06833=1227.317,18.838,-42.416,-179.292,5.372,148.721
C06834=1227.322,18.589,-42.401,-179.294,5.371,148.722
C06835=1227.327,18.340,-42.386,-179.297,5.371,148.722
C06836=1227.332,18.090,-42.371,-179.300,5.370,148.723
C06837=1227.336,17.840,-42.356,-179.302,5.370,148.724
C06838=1227.342,17.591,-42.340,-179.304,5.370,148.724
C06839=1227.347,17.342,-42.325,-179.307,5.369,148.725
C06840=1227.352,17.092,-42.310,-179.310,5.369,148.726
C06841=1227.357,16.843,-42.295,-179.312,5.368,148.727
C06842=1227.362,16.593,-42.279,-179.314,5.369,148.727
C06843=1227.367,16.343,-42.265,-179.317,5.368,148.728
C06844=1227.371,16.094,-42.250,-179.320,5.367,148.729
C06845=1227.377,15.844,-42.234,-179.322,5.367,148.729
C06846=1227.381,15.595,-42.219,-179.325,5.366,148.730
C06847=1227.387,15.345,-42.204,-179.327,5.367,148.731
C06848=1227.392,15.096,-42.189,-179.330,5.366,148.731
C06849=1227.397,14.847,-42.174,-179.332,5.366,148.732
C06850=1227.402,14.597,-42.160,-179.335,5.365,148.733
C06851=1227.407,14.348,-42.145,-179.338,5.365,148.733
C06852=1227.412,14.098,-42.129,-179.340,5.365,148.734
C06853=1227.417,13.849,-42.115,-179.342,5.364,148.735
C06854=1227.422,13.599,-42.099,-179.345,5.364,148.735
C06855=1227.427,13.349,-42.084,-179.348,5.363,148.736
C06856=1227.431,13.100,-42.069,-179.349,5.363,148.737
C06857=1227.437,12.850,-42.054,-179.352,5.363,148.737
C06858=1227.442,12.601,-42.040,-179.354,5.362,148.738
C06859=1227.446,12.352,-42.025,-179.357,5.361,148.739
C06860=1227.452,12.102,-42.010,-179.360,5.361,148.739
C06861=1227.457,11.852,-41.995,-179.362,5.361,148.740
C06862=1227.462,11.603,-41.979,-179.364,5.361,148.741
C06863=1227.467,11.353,-41.965,-179.367,5.360,148.741
C06864=1227.472,11.104,-41.950,-179.370,5.360,148.742
C06865=1227.477,10.854,-41.935,-179.372,5.360,148.743
C06866=1227.482,10.605,-41.920,-179.374,5.359,148.743
C06867=1227.487,10.355,-41.906,-179.377,5.359,148.744
C06868=1227.492,10.106,-41.891,-179.380,5.358,148.745
C06869=1227.497,9.856,-41.876,-179.382,5.358,148.745
C06870=1227.502,9.607,-41.861,-179.385,5.358,148.746
C06871=1227.507,9.358,-41.847,-179.387,5.358,148.747
C06872=1227.512,9.108,-41.831,-179.390,5.357,148.748
C06873=1227.517,8.858,-41.817,-179.392,5.356,148.748
C06874=1227.522,8.609,-41.802,-179.395,5.357,148.749
C06875=1227.527,8.360,-41.787,-179.397,5.356,148.750
C06876=1227.532,8.110,-41.772,-179.400,5.356,148.750
C06877=1227.537,7.860,-41.758,-179.403,5.355,148.751
C06878=1227.542,7.611,-41.743,-179.405,5.355,148.752
C06879=1227.548,7.361,-41.728,-179.407,5.355,148.752
C06880=1227.552,7.112,-41.713,-179.410,5.354,148.753
C06881=1227.557,6.863,-41.698,-179.413,5.354,148.754
C06882=1227.562,6.613,-41.684,-179.415,5.354,148.754
C06883=1227.567,6.363,-41.670,-179.417,5.354,148.755
C06884=1227.572,6.114,-41.654,-179.420,5.353,148.756
C06885=1227.577,5.864,-41.640,-179.423,5.353,148.756
C06886=1227.582,5.615,-41.625,-179.425,5.353,148.757
C06887=1227.587,5.365,-41.611,-179.427,5.352,148.758
C06888=1227.593,5.115,-41.596,-179.430,5.352,148.759
C06889=1227.597,4.866,-41.581,-179.433,5.351,148.759
C06890=1227.602,4.616,-41.567,-179.435,5.352,148.760
C06891=1227.607,4.367,-41.552,-179.437,5.351,148.761
C06892=1227.612,4.118,-41.537,-179.440,5.350,148.761
C06893=1227.618,3.849,-41.521,-179.443,5.350,148.762
C06894=1227.623,3.579,-41.506,-179.445,5.349,148.763
C06895=1227.628,3.310,-41.490,-179.448,5.349,148.764
C06896=1227.634,3.042,-41.475,-179.450,5.350,148.764
C06897=1227.639,2.793,-41.461,-179.453,5.349,148.765
C06898=1227.644,2.543,-41.445,-179.456,5.348,148.766
C06899=1227.649,2.293,-41.431,-179.458,5.348,148.766
C06900=1227.654,2.044,-41.417,-179.461,5.348,148.767
C06901=1227.659,1.794,-41.402,-179.463,5.348,148.768
C06902=1227.664,1.545,-41.387,-179.466,5.347,148.768
C06903=1227.669,1.295,-41.373,-179.468,5.347,148.769
C06904=1227.674,1.045,-41.359,-179.471,5.347,148.770
C06905=1227.679,0.796,-41.344,-179.473,5.346,148.770
C06906=1227.685,0.547,-41.329,-179.476,5.346,148.771
C06907=1227.690,0.297,-41.315,-179.479,5.345,148.772
C06908=1227.695,0.048,-41.301,-179.481,5.346,148.773
C06909=1227.700,-0.202,-41.286,-179.483,5.345,148.773
C06910=1227.705,-0.452,-41.272,-179.486,5.345,148.774
C06911=1227.710,-0.702,-41.258,-179.489,5.344,148.775
C06912=1227.714,-0.951,-41.243,-179.491,5.344,148.775
C06913=1227.719,-1.200,-41.229,-179.493,5.344,148.776
C06914=1227.725,-1.449,-41.215,-179.496,5.343,148.777
C06915=1227.730,-1.699,-41.200,-179.498,5.344,148.777
C06916=1227.735,-1.949,-41.186,-179.501,5.343,148.778
C06917=1227.740,-2.198,-41.172,-179.503,5.343,148.779
C06918=1227.745,-2.448,-41.158,-179.506,5.342,148.779
C06919=1227.749,-2.697,-41.143,-179.508,5.342,148.780
C06920=1227.754,-2.947,-41.128,-179.511,5.342,148.781
C06921=1227.760,-3.196,-41.114,-179.513,5.341,148.781
C06922=1227.765,-3.446,-41.100,-179.515,5.342,148.782
C06923=1227.770,-3.695,-41.086,-179.518,5.341,148.783
C06924=1227.775,-3.945,-41.072,-179.521,5.341,148.784
C06925=1227.779,-4.195,-41.057,-179.523,5.340,148.784
C06926=1227.784,-4.445,-41.043,-179.525,5.340,148.785
C06927=1227.790,-4.694,-41.029,-179.528,5.340,148.786
C06928=1227.795,-4.943,-41.015,-179.531,5.339,148.786
C06929=1227.800,-5.193,-41.001,-179.533,5.339,148.787
C06930=1227.805,-5.443,-40.986,-179.536,5.339,148.788
C06931=1227.810,-5.692,-40.972,-179.538,5.339,148.788
C06932=1227.815,-5.941,-40.958,-179.541,5.338,148.789
C06933=1227.820,-6.191,-40.944,-179.543,5.338,148.790
C06934=1227.825,-6.441,-40.930,-179.546,5.338,148.790
C06935=1227.830,-6.691,-40.915,-179.548,5.337,148.791
C06936=1227.835,-6.940,-40.901,-179.550,5.338,148.792
C06937=1227.841,-7.189,-40.887,-179.553,5.337,148.793
C06938=1227.846,-7.439,-40.873,-179.556,5.337,148.793
C06939=1227.851,-7.689,-40.859,-179.558,5.336,148.794
C06940=1227.856,-7.938,-40.844,-179.560,5.336,148.795
C06941=1227.861,-8.187,-40.830,-179.563,5.336,148.795
C06942=1227.865,-8.437,-40.817,-179.566,5.335,148.796
C06943=1227.870,-8.686,-40.802,-179.568,5.336,148.797
C06944=1227.875,-8.936,-40.788,-179.570,5.335,148.797
C06945=1227.881,-9.185,-40.774,-179.573,5.335,148.798
C06946=1227.886,-9.435,-40.760,-179.576,5.334,148.799
C06947=1227.891,-9.685,-40.746,-179.578,5.334,148.799
C06948=1227.896,-9.934,-40.731,-179.580,5.334,148.800
C06949=1227.901,-10.183,-40.717,-179.583,5.333,148.801
C06950=1227.906,-10.433,-40.704,-179.585,5.334,148.802
C06951=1227.911,-10.683,-40.690,-179.588,5.333,148.802
C06952=1227.916,-10.933,-40.676,-179.590,5.333,148.803
C06953=1227.921,-11.182,-40.662,-179.593,5.333,148.804
C06954=1227.926,-11.432,-40.648,-179.595,5.332,148.804
C06955=1227.931,-11.681,-40.633,-179.598,5.332,148.805
C06956=1227.937,-11.930,-40.620,-179.600,5.332,148.806
C06957=1227.941,-12.180,-40.607,-179.603,5.332,148.806
C06958=1227.946,-12.430,-40.592,-179.605,5.331,148.807
C06959=1227.951,-12.680,-40.578,-179.608,5.331,148.808
C06960=1227.957,-12.929,-40.564,-179.610,5.331,148.808
C06961=1227.962,-13.178,-40.550,-179.613,5.330,148.809
C06962=1227.966,-13.428,-40.537,-179.615,5.330,148.810
C06963=1227.972,-13.677,-40.523,-179.617,5.330,148.811
C06964=1227.977,-13.927,-40.509,-179.620,5.330,148.811
C06965=1227.982,-14.177,-40.494,-179.623,5.329,148.812
C06966=1227.988,-14.426,-40.481,-179.625,5.329,148.813
C06967=1227.992,-14.676,-40.468,-179.627,5.329,148.813
C06968=1227.997,-14.926,-40.453,-179.630,5.328,148.814
C06969=1228.002,-15.175,-40.439,-179.632,5.329,148.815
C06970=1228.008,-15.425,-40.426,-179.635,5.328,148.815
C06971=1228.012,-15.674,-40.412,-179.638,5.328,148.816
C06972=1228.017,-15.923,-40.398,-179.640,5.328,148.817
C06973=1228.023,-16.174,-40.385,-179.642,5.327,148.817
C06974=1228.028,-16.423,-40.370,-179.645,5.327,148.818
C06975=1228.032,-16.672,-40.357,-179.647,5.327,148.819
C06976=1228.037,-16.922,-40.343,-179.650,5.327,148.820
C06977=1228.043,-17.172,-40.329,-179.652,5.326,148.820
C06978=1228.047,-17.421,-40.316,-179.654,5.327,148.821
C06979=1228.052,-17.671,-40.302,-179.657,5.326,148.822
C06980=1228.058,-17.920,-40.288,-179.660,5.326,148.822
C06981=1228.063,-18.170,-40.274,-179.662,5.326,148.823
C06982=1228.068,-18.420,-40.261,-179.664,5.325,148.824
C06983=1228.073,-18.669,-40.247,-179.667,5.325,148.824
C06984=1228.078,-18.919,-40.233,-179.669,5.325,148.825
C06985=1228.083,-19.169,-40.220,-179.672,5.325,148.826
C06986=1228.088,-19.418,-40.206,-179.674,5.324,148.826
C06987=1228.093,-19.667,-40.192,-179.677,5.324,148.827
C06988=1228.098,-19.917,-40.179,-179.679,5.324,148.828
C06989=1228.103,-20.166,-40.165,-179.682,5.323,148.829
C06990=1228.109,-20.416,-40.152,-179.684,5.324,148.829
C06991=1228.113,-20.665,-40.138,-179.687,5.323,148.830
C06992=1228.119,-20.916,-40.124,-179.690,5.323,148.831
C06993=1228.123,-21.164,-40.111,-179.692,5.323,148.832
C06994=1228.129,-21.415,-40.098,-179.695,5.323,148.832
C06995=1228.134,-21.664,-40.084,-179.697,5.322,148.833
C06996=1228.138,-21.913,-40.070,-179.699,5.323,148.834
C06997=1228.144,-22.183,-40.056,-179.702,5.322,148.834
C06998=1228.150,-22.452,-40.041,-179.705,5.322,148.835
C06999=1228.156,-22.721,-40.026,-179.707,5.321,148.836
C07000=1228.160,-22.990,-40.012,-179.710,5.321,148.837
C07001=1228.166,-23.241,-39.998,-179.712,5.321,148.837
C07002=1228.171,-23.490,-39.984,-179.715,5.321,148.838
C07003=1228.176,-23.740,-39.971,-179.717,5.321,148.839
C07004=1228.181,-23.989,-39.957,-179.720,5.321,148.839
C07005=1228.186,-24.239,-39.944,-179.723,5.320,148.840
C07006=1228.192,-24.488,-39.931,-179.725,5.320,148.841
C07007=1228.196,-24.738,-39.918,-179.727,5.320,148.842
C07008=1228.202,-24.987,-39.904,-179.730,5.319,148.842
C07009=1228.206,-25.237,-39.891,-179.732,5.320,148.843
C07010=1228.212,-25.486,-39.877,-179.735,5.319,148.844
C07011=1228.216,-25.736,-39.864,-179.737,5.319,148.844
C07012=1228.222,-25.986,-39.851,-179.739,5.319,148.845
C07013=1228.227,-26.236,-39.837,-179.742,5.319,148.846
C07014=1228.232,-26.485,-39.824,-179.745,5.318,148.846
C07015=1228.237,-26.735,-39.810,-179.747,5.318,148.847
C07016=1228.242,-26.984,-39.797,-179.749,5.318,148.848
C07017=1228.247,-27.234,-39.783,-179.752,5.317,148.849
C07018=1228.252,-27.483,-39.771,-179.754,5.318,148.849
C07019=1228.257,-27.733,-39.756,-179.757,5.317,148.850
C07020=1228.262,-27.982,-39.744,-179.759,5.317,148.851
C07021=1228.268,-28.233,-39.730,-179.762,5.317,148.851
C07022=1228.273,-28.481,-39.717,-179.764,5.316,148.852
C07023=1228.277,-28.731,-39.704,-179.766,5.317,148.853
C07024=1228.283,-28.981,-39.691,-179.769,5.316,148.853
C07025=1228.287,-29.230,-39.677,-179.772,5.316,148.854
C07026=1228.293,-29.480,-39.664,-179.774,5.316,148.855
C07027=1228.298,-29.730,-39.651,-179.776,5.316,148.856
C07028=1228.303,-29.979,-39.637,-179.779,5.315,148.856
C07029=1228.308,-30.229,-39.624,-179.781,5.315,148.857
C07030=1228.313,-30.479,-39.611,-179.784,5.315,148.858
C07031=1228.319,-30.728,-39.598,-179.786,5.315,148.858
C07032=1228.323,-30.977,-39.585,-179.789,5.315,148.859
C07033=1228.329,-31.227,-39.571,-179.791,5.314,148.860
C07034=1228.333,-31.477,-39.558,-179.793,5.315,148.860
C07035=1228.339,-31.727,-39.545,-179.796,5.314,148.861
C07036=1228.343,-31.976,-39.531,-179.799,5.314,148.862
C07037=1228.348,-32.225,-39.519,-179.801,5.314,148.863
C07038=1228.354,-32.476,-39.505,-179.804,5.314,148.863
C07039=1228.359,-32.725,-39.493,-179.806,5.314,148.864
C07040=1228.365,-32.975,-39.480,-179.809,5.314,148.865
C07041=1228.369,-33.224,-39.466,-179.811,5.313,148.866
C07042=1228.374,-33.473,-39.453,-179.813,5.313,148.866
C07043=1228.379,-33.724,-39.440,-179.816,5.313,148.867
C07044=1228.384,-33.973,-39.427,-179.819,5.312,148.868
C07045=1228.390,-34.222,-39.414,-179.821,5.313,148.868
C07046=1228.395,-34.473,-39.401,-179.823,5.312,148.869
C07047=1228.400,-34.721,-39.388,-179.826,5.312,148.870
C07048=1228.404,-34.971,-39.375,-179.828,5.312,148.870
C07049=1228.410,-35.221,-39.361,-179.831,5.312,148.871
C07050=1228.415,-35.470,-39.349,-179.833,5.312,148.872
C07051=1228.420,-35.720,-39.336,-179.836,5.311,148.873
C07052=1228.425,-35.970,-39.323,-179.838,5.311,148.873
C07053=1228.431,-36.219,-39.310,-179.840,5.311,148.874
C07054=1228.435,-36.469,-39.297,-179.843,5.311,148.875
C07055=1228.441,-36.718,-39.283,-179.845,5.311,148.875
C07056=1228.446,-36.968,-39.271,-179.848,5.310,148.876
C07057=1228.450,-37.218,-39.258,-179.850,5.310,148.877
C07058=1228.456,-37.467,-39.244,-179.853,5.310,148.877
C07059=1228.461,-37.717,-39.231,-179.855,5.310,148.878
C07060=1228.466,-37.967,-39.219,-179.857,5.310,148.879
C07061=1228.471,-38.216,-39.206,-179.860,5.310,148.880
C07062=1228.476,-38.466,-39.193,-179.863,5.309,148.880
C07063=1228.481,-38.716,-39.180,-179.865,5.309,148.881
C07064=1228.486,-38.965,-39.168,-179.867,5.309,148.882
C07065=1228.492,-39.215,-39.154,-179.869,5.309,148.882
C07066=1228.497,-39.465,-39.141,-179.872,5.309,148.883
C07067=1228.502,-39.714,-39.129,-179.875,5.308,148.884
C07068=1228.507,-39.963,-39.116,-179.877,5.309,148.884
C07069=1228.512,-40.213,-39.103,-179.879,5.308,148.885
C07070=1228.517,-40.463,-39.090,-179.882,5.308,148.886
C07071=1228.523,-40.712,-39.077,-179.884,5.308,148.887
C07072=1228.527,-40.962,-39.064,-179.887,5.307,148.887
C07073=1228.532,-41.211,-39.052,-179.889,5.308,148.888
C07074=1228.537,-41.461,-39.039,-179.892,5.307,148.889
C07075=1228.543,-41.711,-39.026,-179.894,5.308,148.889
C07076=1228.548,-41.960,-39.013,-179.896,5.307,148.890
C07077=1228.553,-42.210,-39.000,-179.900,5.307,148.891
C07078=1228.557,-42.460,-38.987,-179.902,5.307,148.892
C07079=1228.563,-42.710,-38.976,-179.904,5.307,148.892
C07080=1228.569,-42.959,-38.962,-179.906,5.307,148.893
C07081=1228.574,-43.209,-38.950,-179.909,5.307,148.894
C07082=1228.578,-43.459,-38.937,-179.912,5.306,148.894
C07083=1228.583,-43.708,-38.924,-179.914,5.307,148.895
C07084=1228.589,-43.957,-38.912,-179.916,5.306,148.896
C07085=1228.594,-44.207,-38.899,-179.919,5.306,148.897
C07086=1228.598,-44.457,-38.886,-179.921,5.306,148.897
C07087=1228.604,-44.706,-38.873,-179.924,5.305,148.898
C07088=1228.610,-44.956,-38.861,-179.926,5.306,148.899
C07089=1228.615,-45.206,-38.848,-179.929,5.305,148.899
C07090=1228.619,-45.456,-38.835,-179.931,5.306,148.900
C07091=1228.624,-45.705,-38.823,-179.933,5.305,148.901
C07092=1228.629,-45.954,-38.810,-179.936,5.305,148.901
C07093=1228.635,-46.204,-38.798,-179.938,5.305,148.902
C07094=1228.639,-46.454,-38.785,-179.941,5.304,148.903
C07095=1228.645,-46.704,-38.772,-179.943,5.305,148.904
C07096=1228.650,-46.953,-38.760,-179.946,5.304,148.904
C07097=1228.655,-47.202,-38.747,-179.948,5.304,148.905
C07098=1228.661,-47.452,-38.735,-179.950,5.304,148.906
C07099=1228.665,-47.702,-38.722,-179.953,5.304,148.906
C07100=1228.671,-47.952,-38.710,-179.955,5.304,148.907
C07101=1228.676,-48.221,-38.696,-179.958,5.303,148.908
C07102=1228.682,-48.491,-38.683,-179.961,5.303,148.909
C07103=1228.687,-48.761,-38.669,-179.963,5.304,148.909
C07104=1228.693,-49.030,-38.656,-179.966,5.303,148.910
C07105=1228.698,-49.281,-38.643,-179.968,5.303,148.911
C07106=1228.703,-49.530,-38.631,-179.970,5.303,148.912
C07107=1228.708,-49.779,-38.618,-179.973,5.303,148.912
C07108=1228.713,-50.029,-38.606,-179.975,5.303,148.913
C07109=1228.718,-50.279,-38.594,-179.978,5.302,148.914
C07110=1228.723,-50.529,-38.581,-179.980,5.302,148.914
C07111=1228.728,-50.778,-38.568,-179.983,5.302,148.915
C07112=1228.734,-51.028,-38.556,-179.985,5.302,148.916
C07113=1228.739,-51.277,-38.544,-179.987,5.302,148.916
C07114=1228.744,-51.527,-38.531,-179.990,5.302,148.917
C07115=1228.749,-51.776,-38.519,-179.992,5.302,148.918
C07116=1228.754,-52.026,-38.506,-179.995,5.301,148.919
C07117=1228.759,-52.276,-38.494,-179.997,5.301,148.919
C07118=1228.764,-52.526,-38.482,-179.999,5.301,148.920
C07119=1228.769,-52.775,-38.469,179.998,5.301,148.921
C07120=1228.775,-53.025,-38.457,179.996,5.301,148.921
C07121=1228.780,-53.274,-38.445,179.993,5.301,148.922
C07122=1228.785,-53.524,-38.432,179.991,5.301,148.923
C07123=1228.790,-53.774,-38.420,179.988,5.301,148.924
C07124=1228.795,-54.024,-38.407,179.985,5.300,148.924
C07125=1228.800,-54.274,-38.395,179.983,5.301,148.925
C07126=1228.806,-54.523,-38.383,179.980,5.300,148.926
C07127=1228.811,-54.772,-38.370,179.978,5.301,148.927
C07128=1228.816,-55.022,-38.358,179.976,5.300,148.927
C07129=1228.821,-55.271,-38.346,179.974,5.300,148.928
C07130=1228.826,-55.521,-38.334,179.971,5.300,148.929
C07131=1228.830,-55.771,-38.321,179.968,5.299,148.929
C07132=1228.836,-56.021,-38.309,179.966,5.300,148.930
C07133=1228.841,-56.270,-38.297,179.964,5.299,148.931
C07134=1228.846,-56.520,-38.285,179.961,5.300,148.931
C07135=1228.852,-56.770,-38.272,179.959,5.299,148.932
C07136=1228.857,-57.020,-38.260,179.957,5.300,148.933
C07137=1228.862,-57.269,-38.248,179.954,5.299,148.934
C07138=1228.867,-57.518,-38.237,179.952,5.299,148.934
C07139=1228.872,-57.768,-38.224,179.949,5.299,148.935
C07140=1228.877,-58.018,-38.212,179.947,5.298,148.936
C07141=1228.883,-58.267,-38.200,179.944,5.299,148.936
C07142=1228.888,-58.517,-38.188,179.942,5.298,148.937
C07143=1228.892,-58.767,-38.175,179.940,5.299,148.938
C07144=1228.897,-59.017,-38.163,179.937,5.298,148.939
C07145=1228.902,-59.266,-38.151,179.935,5.298,148.939
C07146=1228.908,-59.516,-38.139,179.932,5.298,148.940
C07147=1228.913,-59.766,-38.127,179.930,5.298,148.941
C07148=1228.918,-60.015,-38.114,179.928,5.298,148.941
C07149=1228.924,-60.265,-38.103,179.925,5.297,148.942
C07150=1228.928,-60.514,-38.091,179.923,5.298,148.943
C07151=1228.934,-60.764,-38.079,179.920,5.297,148.943
C07152=1228.939,-61.014,-38.067,179.918,5.298,148.944
C07153=1228.944,-61.263,-38.054,179.915,5.297,148.945
C07154=1228.949,-61.513,-38.042,179.913,5.297,148.946
C07155=1228.954,-61.762,-38.030,179.911,5.297,148.946
C07156=1228.959,-62.012,-38.018,179.909,5.297,148.947
C07157=1228.965,-62.262,-38.006,179.906,5.297,148.948
C07158=1228.970,-62.511,-37.994,179.904,5.297,148.948
C07159=1228.975,-62.761,-37.983,179.901,5.297,148.949
C07160=1228.980,-63.011,-37.971,179.898,5.296,148.950
C07161=1228.985,-63.260,-37.958,179.896,5.297,148.951
C07162=1228.991,-63.510,-37.946,179.894,5.296,148.951
C07163=1228.995,-63.760,-37.935,179.892,5.296,148.952
C07164=1229.001,-64.010,-37.923,179.889,5.296,148.953
C07165=1229.006,-64.259,-37.910,179.887,5.296,148.953
C07166=1229.011,-64.509,-37.899,179.884,5.296,148.954
C07167=1229.016,-64.759,-37.887,179.882,5.296,148.955
C07168=1229.021,-65.008,-37.875,179.879,5.296,148.955
C07169=1229.026,-65.258,-37.863,179.877,5.296,148.956
C07170=1229.031,-65.508,-37.851,179.875,5.296,148.957
C07171=1229.037,-65.757,-37.840,179.872,5.295,148.958
C07172=1229.042,-66.007,-37.827,179.870,5.295,148.958
C07173=1229.047,-66.257,-37.815,179.867,5.295,148.959
C07174=1229.052,-66.506,-37.804,179.865,5.295,148.960
C07175=1229.057,-66.756,-37.792,179.862,5.295,148.960
C07176=1229.062,-67.006,-37.779,179.860,5.295,148.961
C07177=1229.067,-67.255,-37.768,179.858,5.295,148.962
C07178=1229.072,-67.505,-37.756,179.856,5.295,148.963
C07179=1229.078,-67.755,-37.744,179.853,5.295,148.963
C07180=1229.083,-68.004,-37.733,179.851,5.295,148.964
C07181=1229.089,-68.254,-37.721,179.848,5.294,148.965
C07182=1229.094,-68.503,-37.709,179.846,5.295,148.965
C07183=1229.098,-68.753,-37.698,179.843,5.294,148.966
C07184=1229.104,-69.003,-37.686,179.841,5.294,148.967
C07185=1229.109,-69.252,-37.674,179.839,5.294,148.967
C07186=1229.114,-69.502,-37.663,179.836,5.294,148.968
C07187=1229.119,-69.752,-37.651,179.834,5.294,148.969
C07188=1229.124,-70.001,-37.639,179.831,5.294,148.970
C07189=1229.129,-70.251,-37.627,179.829,5.294,148.970
C07190=1229.135,-70.501,-37.615,179.826,5.293,148.971
C07191=1229.140,-70.750,-37.604,179.824,5.294,148.972
C07192=1229.145,-71.000,-37.592,179.822,5.293,148.972
C07193=1229.150,-71.250,-37.581,179.820,5.294,148.973
C07194=1229.156,-71.500,-37.569,179.817,5.293,148.974
C07195=1229.161,-71.750,-37.557,179.815,5.294,148.975
C07196=1229.166,-71.999,-37.546,179.812,5.293,148.975
C07197=1229.171,-72.249,-37.534,179.810,5.293,148.976
C07198=1229.176,-72.499,-37.523,179.807,5.293,148.977
C07199=1229.182,-72.748,-37.511,179.805,5.293,148.977
C07200=1229.186,-72.997,-37.499,179.803,5.293,148.978
C07201=1229.192,-73.247,-37.487,179.801,5.293,148.979
C07202=1229.196,-73.497,-37.476,179.798,5.293,148.980
C07203=1229.202,-73.746,-37.464,179.795,5.292,148.980
C07204=1229.207,-73.996,-37.452,179.793,5.293,148.981
C07205=1229.213,-74.267,-37.440,179.791,5.292,148.982
C07206=1229.218,-74.537,-37.428,179.788,5.293,148.983
C07207=1229.224,-74.808,-37.416,179.785,5.292,148.983
C07208=1229.229,-75.077,-37.403,179.783,5.292,148.984
C07209=1229.235,-75.327,-37.391,179.780,5.292,148.985
C07210=1229.240,-75.577,-37.380,179.778,5.292,148.985
C07211=1229.245,-75.827,-37.368,179.776,5.292,148.986
C07212=1229.250,-76.077,-37.357,179.773,5.292,148.987
C07213=1229.256,-76.326,-37.345,179.771,5.292,148.988
C07214=1229.260,-76.575,-37.334,179.768,5.292,148.988
C07215=1229.266,-76.825,-37.322,179.766,5.292,148.989
C07216=1229.271,-77.075,-37.311,179.764,5.292,148.990
C07217=1229.276,-77.325,-37.299,179.761,5.292,148.990
C07218=1229.282,-77.574,-37.289,179.759,5.291,148.991
C07219=1229.287,-77.824,-37.277,179.757,5.292,148.992
C07220=1229.292,-78.074,-37.265,179.754,5.291,148.993
C07221=1229.297,-78.324,-37.253,179.752,5.292,148.993
C07222=1229.302,-78.574,-37.242,179.749,5.291,148.994
C07223=1229.307,-78.822,-37.231,179.747,5.292,148.995
C07224=1229.313,-79.072,-37.219,179.744,5.291,148.995
C07225=1229.317,-79.322,-37.208,179.742,5.291,148.996
C07226=1229.323,-79.572,-37.196,179.740,5.291,148.997
C07227=1229.328,-79.822,-37.186,179.738,5.291,148.997
C07228=1229.334,-80.071,-37.174,179.735,5.291,148.998
C07229=1229.338,-80.321,-37.163,179.733,5.291,148.999
C07230=1229.343,-80.571,-37.152,179.730,5.291,149.000
C07231=1229.349,-80.821,-37.140,179.728,5.291,149.000
C07232=1229.354,-81.070,-37.129,179.725,5.291,149.001
C07233=1229.360,-81.320,-37.118,179.723,5.291,149.002
C07234=1229.364,-81.570,-37.106,179.721,5.291,149.002
C07235=1229.369,-81.819,-37.095,179.719,5.291,149.003
C07236=1229.375,-82.069,-37.083,179.716,5.290,149.004
C07237=1229.380,-82.318,-37.072,179.714,5.291,149.005
C07238=1229.385,-82.568,-37.062,179.711,5.290,149.005
C07239=1229.390,-82.818,-37.050,179.708,5.290,149.006
C07240=1229.395,-83.067,-37.039,179.706,5.290,149.007
C07241=1229.400,-83.317,-37.027,179.704,5.290,149.007
C07242=1229.406,-83.568,-37.016,179.702,5.290,149.008
C07243=1229.411,-83.817,-37.005,179.699,5.290,149.009
C07244=1229.416,-84.066,-36.994,179.697,5.290,149.010
C07245=1229.421,-84.316,-36.982,179.694,5.290,149.010
C07246=1229.426,-84.566,-36.972,179.692,5.290,149.011
C07247=1229.432,-84.815,-36.961,179.689,5.289,149.012
C07248=1229.437,-85.065,-36.949,179.687,5.290,149.012
C07249=1229.442,-85.315,-36.938,179.685,5.289,149.013
C07250=1229.447,-85.565,-36.927,179.683,5.290,149.014
C07251=1229.453,-85.814,-36.915,179.680,5.289,149.015
C07252=1229.457,-86.064,-36.904,179.678,5.289,149.015
C07253=1229.462,-86.314,-36.894,179.676,5.289,149.016
C07254=1229.468,-86.563,-36.883,179.674,5.289,149.016
C07255=1229.473,-86.813,-36.871,179.671,5.289,149.017
C07256=1229.478,-87.063,-36.860,179.669,5.289,149.018
C07257=1229.483,-87.312,-36.849,179.666,5.289,149.019
C07258=1229.488,-87.562,-36.838,179.664,5.289,149.019
C07259=1229.494,-87.812,-36.827,179.661,5.288,149.020
C07260=1229.499,-88.061,-36.816,179.659,5.289,149.021
C07261=1229.504,-88.311,-36.805,179.657,5.289,149.021
C07262=1229.509,-88.561,-36.794,179.654,5.289,149.022
C07263=1229.515,-88.810,-36.782,179.652,5.289,149.023
C07264=1229.520,-89.061,-36.772,179.650,5.289,149.024
C07265=1229.524,-89.310,-36.761,179.648,5.289,149.024
C07266=1229.530,-89.560,-36.750,179.645,5.289,149.025
C07267=1229.536,-89.810,-36.739,179.643,5.289,149.026
C07268=1229.540,-90.059,-36.727,179.640,5.288,149.026
C07269=1229.546,-90.309,-36.717,179.638,5.289,149.027
C07270=1229.550,-90.558,-36.706,179.635,5.288,149.028
C07271=1229.555,-90.809,-36.695,179.633,5.289,149.028
C07272=1229.562,-91.058,-36.684,179.631,5.288,149.029
C07273=1229.567,-91.308,-36.673,179.629,5.289,149.030
C07274=1229.572,-91.557,-36.662,179.626,5.288,149.031
C07275=1229.577,-91.807,-36.652,179.624,5.289,149.031
C07276=1229.582,-92.057,-36.640,179.621,5.288,149.032
C07277=1229.588,-92.307,-36.629,179.619,5.288,149.033
C07278=1229.593,-92.556,-36.618,179.616,5.288,149.033
C07279=1229.598,-92.806,-36.608,179.614,5.288,149.034
C07280=1229.603,-93.056,-36.597,179.612,5.288,149.035
C07281=1229.608,-93.306,-36.586,179.610,5.288,149.035
C07282=1229.613,-93.555,-36.575,179.607,5.287,149.036
C07283=1229.618,-93.805,-36.565,179.605,5.288,149.037
C07284=1229.624,-94.054,-36.553,179.603,5.287,149.038
C07285=1229.629,-94.305,-36.543,179.600,5.288,149.038
C07286=1229.634,-94.554,-36.531,179.598,5.287,149.039
C07287=1229.639,-94.804,-36.521,179.596,5.288,149.040
C07288=1229.644,-95.053,-36.510,179.593,5.287,149.040
C07289=1229.650,-95.303,-36.500,179.591,5.288,149.041
C07290=1229.655,-95.553,-36.489,179.588,5.287,149.042
C07291=1229.660,-95.802,-36.478,179.586,5.287,149.043
C07292=1229.665,-96.052,-36.467,179.583,5.287,149.043
C07293=1229.670,-96.302,-36.456,179.581,5.287,149.044
C07294=1229.676,-96.552,-36.445,179.579,5.287,149.045
C07295=1229.681,-96.802,-36.435,179.577,5.287,149.045
C07296=1229.686,-97.051,-36.424,179.574,5.287,149.046
C07297=1229.691,-97.301,-36.413,179.572,5.287,149.047
C07298=1229.697,-97.550,-36.402,179.570,5.288,149.047
